LIN {X 0,Y 490.023,Z 695.478,A -85,B 0,C 180,E1 -6692.2,E2 -6692.2} C_VEL
LIN {X 0,Y 489.637,Z 706.697,A -85,B 0,C 180,E1 -6693.054,E2 -6693.054} C_VEL
LIN {X 0,Y 489.247,Z 716.032,A -85,B 0,C 180,E1 -6693.937,E2 -6693.937} C_VEL
LIN {X 0,Y 488.869,Z 726.03,A -85,B 0,C 180,E1 -6695.103,E2 -6695.103} C_VEL
LIN {X 0,Y 488.534,Z 734.515,A -85,B 0,C 180,E1 -6696.331,E2 -6696.331} C_VEL
LIN {X 0,Y 488.289,Z 741.806,A -85,B 0,C 180,E1 -6697.663,E2 -6697.663} C_VEL
LIN {X 0,Y 488.104,Z 747.453,A -85,B 0,C 180,E1 -6698.966,E2 -6698.966} C_VEL
LIN {X 0,Y 487.973,Z 752.212,A -85,B 0,C 180,E1 -6700.399,E2 -6700.399} C_VEL
LIN {X 0,Y 487.929,Z 754.875,A -85,B 0,C 180,E1 -6701.497,E2 -6701.497} C_VEL
LIN {X 0,Y 487.873,Z 756.978,A -85,B 0,C 180,E1 -6702.72,E2 -6702.72} C_VEL
LIN {X 0,Y 487.815,Z 758.178,A -85,B 0,C 180,E1 -6703.916,E2 -6703.916} C_VEL
LIN {X 0,Y 487.843,Z 758.558,A -85,B 0,C 180,E1 -6705.097,E2 -6705.097} C_VEL
LIN {X 0,Y 487.798,Z 758.129,A -85,B 0,C 180,E1 -6706.246,E2 -6706.246} C_VEL
LIN {X 0,Y 487.859,Z 756.943,A -85,B 0,C 180,E1 -6707.385,E2 -6707.385} C_VEL
LIN {X 0,Y 487.942,Z 753.839,A -85,B 0,C 180,E1 -6709.053,E2 -6709.053} C_VEL
LIN {X 0,Y 488.009,Z 750.6,A -85,B 0,C 180,E1 -6710.221,E2 -6710.221} C_VEL
LIN {X 0,Y 488.153,Z 746.364,A -85,B 0,C 180,E1 -6711.396,E2 -6711.396} C_VEL
LIN {X 0,Y 488.318,Z 739.847,A -85,B 0,C 180,E1 -6712.809,E2 -6712.809} C_VEL
LIN {X 0,Y 488.606,Z 732.16,A -85,B 0,C 180,E1 -6714.116,E2 -6714.116} C_VEL
LIN {X 0,Y 488.927,Z 724.156,A -85,B 0,C 180,E1 -6715.219,E2 -6715.219} C_VEL
LIN {X 0,Y 489.04,Z 721.727,A -85,B 0,C 180,E1 -6715.512,E2 -6715.512} C_VEL
LIN {X 0,Y 488.548,Z 717.585,A -85,B 0,C 180,E1 -6715.998,E2 -6715.998} C_VEL
LIN {X 0,Y 486.035,Z 710.622,A -85,B 0,C 180,E1 -6716.77,E2 -6716.77} C_VEL
LIN {X 0,Y 483.52,Z 703.21,A -85,B 0,C 180,E1 -6717.488,E2 -6717.488} C_VEL
LIN {X 0,Y 483.027,Z 698.288,A -85,B 0,C 180,E1 -6717.882,E2 -6717.882} C_VEL
LIN {X 0,Y 483.462,Z 686.391,A -85,B 0,C 180,E1 -6718.646,E2 -6718.646} C_VEL
LIN {X 0,Y 483.818,Z 674.44,A -85,B 0,C 180,E1 -6719.224,E2 -6719.224} C_VEL
LIN {X 0,Y 483.703,Z 669.212,A -85,B 0,C 180,E1 -6719.433,E2 -6719.433} C_VEL
LIN {X 0,Y 481.382,Z 657.052,A -85,B 0,C 180,E1 -6719.872,E2 -6719.872} C_VEL
LIN {X 0,Y 480.883,Z 654.653,A -85,B 0,C 180,E1 -6719.948,E2 -6719.948} C_VEL
LIN {X 0,Y 480.973,Z 649.74,A -85,B 0,C 180,E1 -6723.065,E2 -6723.065} C_VEL
LIN {X 0,Y 481.009,Z 645.406,A -85,B 0,C 180,E1 -6725.851,E2 -6725.851} C_VEL
LIN {X 0,Y 481.143,Z 641.233,A -85,B 0,C 180,E1 -6728.582,E2 -6728.582} C_VEL
LIN {X 0,Y 481.289,Z 636.602,A -85,B 0,C 180,E1 -6731.652,E2 -6731.652} C_VEL
LIN {X 0,Y 481.411,Z 632.002,A -85,B 0,C 180,E1 -6734.765,E2 -6734.765} C_VEL
LIN {X 0,Y 481.586,Z 627.011,A -85,B 0,C 180,E1 -6738.211,E2 -6738.211} C_VEL
LIN {X 0,Y 481.544,Z 624.616,A -85,B 0,C 180,E1 -6739.913,E2 -6739.913} C_VEL
LIN {X 0,Y 481.85,Z 624.467,A -85,B 0,C 180,E1 -6742.664,E2 -6742.664} C_VEL
LIN {X 0,Y 481.783,Z 624.475,A -85,B 0,C 180,E1 -6744.978,E2 -6744.978} C_VEL
LIN {X 0,Y 481.932,Z 624.454,A -85,B 0,C 180,E1 -6747.492,E2 -6747.492} C_VEL
LIN {X 0,Y 481.91,Z 624.46,A -85,B 0,C 180,E1 -6750.835,E2 -6750.835} C_VEL
LIN {X 0,Y 481.932,Z 624.455,A -85,B 0,C 180,E1 -6752.507,E2 -6752.507} C_VEL
LIN {X 0,Y 481.811,Z 624.469,A -85,B 0,C 180,E1 -6755.86,E2 -6755.86} C_VEL
LIN {X 0,Y 481.708,Z 624.483,A -85,B 0,C 180,E1 -6758.389,E2 -6758.389} C_VEL
LIN {X 0,Y 481.338,Z 624.586,A -85,B 0,C 180,E1 -6761.154,E2 -6761.154} C_VEL
LIN {X 0,Y 481.208,Z 629.999,A -85,B 0,C 180,E1 -6764.375,E2 -6764.375} C_VEL
LIN {X 0,Y 481.122,Z 634.354,A -85,B 0,C 180,E1 -6766.986,E2 -6766.986} C_VEL
LIN {X 0,Y 481.049,Z 638.759,A -85,B 0,C 180,E1 -6769.634,E2 -6769.634} C_VEL
LIN {X 0,Y 480.996,Z 643.209,A -85,B 0,C 180,E1 -6772.327,E2 -6772.327} C_VEL
LIN {X 0,Y 480.957,Z 647.726,A -85,B 0,C 180,E1 -6775.072,E2 -6775.072} C_VEL
LIN {X 0,Y 480.865,Z 652.373,A -85,B 0,C 180,E1 -6777.884,E2 -6777.884} C_VEL
LIN {X 0,Y 480.892,Z 654.41,A -85,B 0,C 180,E1 -6779.133,E2 -6779.133} C_VEL
LIN {X 0,Y 483.713,Z 669.153,A -85,B 0,C 180,E1 -6779.663,E2 -6779.663} C_VEL
LIN {X 0,Y 483.735,Z 677.755,A -85,B 0,C 180,E1 -6780.021,E2 -6780.021} C_VEL
LIN {X 0,Y 483.363,Z 688.737,A -85,B 0,C 180,E1 -6780.589,E2 -6780.589} C_VEL
LIN {X 0,Y 482.887,Z 700.545,A -85,B 0,C 180,E1 -6781.385,E2 -6781.385} C_VEL
LIN {X 0,Y 482.421,Z 711.603,A -85,B 0,C 180,E1 -6782.332,E2 -6782.332} C_VEL
LIN {X 0,Y 481.997,Z 721.578,A -85,B 0,C 180,E1 -6783.396,E2 -6783.396} C_VEL
LIN {X 0,Y 481.589,Z 731.3,A -85,B 0,C 180,E1 -6784.69,E2 -6784.69} C_VEL
LIN {X 0,Y 481.293,Z 738.762,A -85,B 0,C 180,E1 -6785.94,E2 -6785.94} C_VEL
LIN {X 0,Y 481.113,Z 744.188,A -85,B 0,C 180,E1 -6787.054,E2 -6787.054} C_VEL
LIN {X 0,Y 480.98,Z 749.367,A -85,B 0,C 180,E1 -6788.388,E2 -6788.388} C_VEL
LIN {X 0,Y 480.842,Z 753.003,A -85,B 0,C 180,E1 -6789.598,E2 -6789.598} C_VEL
LIN {X 0,Y 480.715,Z 756.291,A -85,B 0,C 180,E1 -6791.139,E2 -6791.139} C_VEL
LIN {X 0,Y 480.714,Z 757.779,A -85,B 0,C 180,E1 -6792.261,E2 -6792.261} C_VEL
LIN {X 0,Y 480.698,Z 758.562,A -85,B 0,C 180,E1 -6793.405,E2 -6793.405} C_VEL
LIN {X 0,Y 480.749,Z 758.608,A -85,B 0,C 180,E1 -6794.563,E2 -6794.563} C_VEL
LIN {X 0,Y 480.737,Z 757.873,A -85,B 0,C 180,E1 -6795.752,E2 -6795.752} C_VEL
LIN {X 0,Y 480.748,Z 756.287,A -85,B 0,C 180,E1 -6796.965,E2 -6796.965} C_VEL
LIN {X 0,Y 480.85,Z 753.79,A -85,B 0,C 180,E1 -6798.193,E2 -6798.193} C_VEL
LIN {X 0,Y 480.972,Z 750.253,A -85,B 0,C 180,E1 -6799.448,E2 -6799.448} C_VEL
LIN {X 0,Y 481.131,Z 745.519,A -85,B 0,C 180,E1 -6800.73,E2 -6800.73} C_VEL
LIN {X 0,Y 481.281,Z 739.339,A -85,B 0,C 180,E1 -6802.049,E2 -6802.049} C_VEL
LIN {X 0,Y 481.631,Z 731.527,A -85,B 0,C 180,E1 -6803.375,E2 -6803.375} C_VEL
LIN {X 0,Y 481.975,Z 722.802,A -85,B 0,C 180,E1 -6804.555,E2 -6804.555} C_VEL
LIN {X 0,Y 482.375,Z 713.597,A -85,B 0,C 180,E1 -6805.571,E2 -6805.571} C_VEL
LIN {X 0,Y 482.775,Z 704.293,A -85,B 0,C 180,E1 -6806.414,E2 -6806.414} C_VEL
LIN {X 0,Y 483.225,Z 692.734,A -85,B 0,C 180,E1 -6807.258,E2 -6807.258} C_VEL
LIN {X 0,Y 483.693,Z 679.943,A -85,B 0,C 180,E1 -6807.971,E2 -6807.971} C_VEL
LIN {X 0,Y 483.839,Z 670.339,A -85,B 0,C 180,E1 -6808.38,E2 -6808.38} C_VEL
LIN {X 0,Y 481.643,Z 658.099,A -85,B 0,C 180,E1 -6808.832,E2 -6808.832} C_VEL
LIN {X 0,Y 480.9,Z 654.64,A -85,B 0,C 180,E1 -6808.931,E2 -6808.931} C_VEL
LIN {X 0,Y 480.927,Z 649.312,A -85,B 0,C 180,E1 -6812.119,E2 -6812.119} C_VEL
LIN {X 0,Y 480.987,Z 644.59,A -85,B 0,C 180,E1 -6814.946,E2 -6814.946} C_VEL
LIN {X 0,Y 481.024,Z 639.996,A -85,B 0,C 180,E1 -6817.674,E2 -6817.674} C_VEL
LIN {X 0,Y 481.088,Z 635.435,A -85,B 0,C 180,E1 -6820.367,E2 -6820.367} C_VEL
LIN {X 0,Y 481.139,Z 630.754,A -85,B 0,C 180,E1 -6823.014,E2 -6823.014} C_VEL
LIN {X 0,Y 481.185,Z 626.098,A -85,B 0,C 180,E1 -6825.623,E2 -6825.623} C_VEL
LIN {X 0,Y 481.186,Z 624.552,A -85,B 0,C 180,E1 -6826.486,E2 -6826.486} C_VEL
LIN {X 0,Y 481.553,Z 624.504,A -85,B 0,C 180,E1 -6828.21,E2 -6828.21} C_VEL
LIN {X 0,Y 481.729,Z 624.482,A -85,B 0,C 180,E1 -6830.765,E2 -6830.765} C_VEL
LIN {X 0,Y 481.786,Z 624.476,A -85,B 0,C 180,E1 -6833.298,E2 -6833.298} C_VEL
LIN {X 0,Y 481.661,Z 624.49,A -85,B 0,C 180,E1 -6835.816,E2 -6835.816} C_VEL
LIN {X 0,Y 481.926,Z 624.456,A -85,B 0,C 180,E1 -6837.492,E2 -6837.492} C_VEL
LIN {X 0,Y 481.937,Z 624.455,A -85,B 0,C 180,E1 -6840,E2 -6840} C_VEL
LIN {X 0,Y 481.925,Z 624.458,A -85,B 0,C 180,E1 -6842.507,E2 -6842.507} C_VEL
LIN {X 0,Y 481.814,Z 624.47,A -85,B 0,C 180,E1 -6845.86,E2 -6845.86} C_VEL
LIN {X 0,Y 481.761,Z 624.477,A -85,B 0,C 180,E1 -6848.388,E2 -6848.388} C_VEL
LIN {X 0,Y 481.749,Z 624.478,A -85,B 0,C 180,E1 -6851.785,E2 -6851.785} C_VEL
LIN {X 0,Y 481.739,Z 624.479,A -85,B 0,C 180,E1 -6855.224,E2 -6855.224} C_VEL
LIN {X 0,Y 481.709,Z 624.484,A -85,B 0,C 180,E1 -6858.722,E2 -6858.722} C_VEL
LIN {X 0,Y 481.644,Z 624.49,A -85,B 0,C 180,E1 -6861.395,E2 -6861.395} C_VEL
LIN {X 0,Y 481.674,Z 624.488,A -85,B 0,C 180,E1 -6864.113,E2 -6864.113} C_VEL
LIN {X 0,Y 481.749,Z 624.48,A -85,B 0,C 180,E1 -6867.141,E2 -6867.141} C_VEL
LIN {X 0,Y 481.685,Z 624.486,A -85,B 0,C 180,E1 -6869.741,E2 -6869.741} C_VEL
LIN {X 0,Y 481.67,Z 624.487,A -85,B 0,C 180,E1 -6872.674,E2 -6872.674} C_VEL
LIN {X 0,Y 481.639,Z 624.491,A -85,B 0,C 180,E1 -6875.71,E2 -6875.71} C_VEL
LIN {X 0,Y 481.669,Z 624.488,A -85,B 0,C 180,E1 -6878.859,E2 -6878.859} C_VEL
LIN {X 0,Y 481.65,Z 624.489,A -85,B 0,C 180,E1 -6881.913,E2 -6881.913} C_VEL
LIN {X 0,Y 481.657,Z 624.491,A -85,B 0,C 180,E1 -6884.458,E2 -6884.458} C_VEL
LIN {X 0,Y 481.646,Z 624.492,A -85,B 0,C 180,E1 -6887.84,E2 -6887.84} C_VEL
LIN {X 0,Y 481.69,Z 624.487,A -85,B 0,C 180,E1 -6891.198,E2 -6891.198} C_VEL
LIN {X 0,Y 482.525,Z 629.808,A -85,B 0,C 180,E1 -6893.852,E2 -6893.852} C_VEL
LIN {X 0,Y 482.49,Z 634.708,A -85,B 0,C 180,E1 -6896.127,E2 -6896.127} C_VEL
LIN {X 0,Y 482.181,Z 641.908,A -85,B 0,C 180,E1 -6899.327,E2 -6899.327} C_VEL
LIN {X 0,Y 481.924,Z 648.538,A -85,B 0,C 180,E1 -6902.183,E2 -6902.183} C_VEL
LIN {X 0,Y 481.664,Z 656.3,A -85,B 0,C 180,E1 -6905.428,E2 -6905.428} C_VEL
LIN {X 0,Y 481.461,Z 664.091,A -85,B 0,C 180,E1 -6908.597,E2 -6908.597} C_VEL
LIN {X 0,Y 481.272,Z 671.804,A -85,B 0,C 180,E1 -6911.658,E2 -6911.658} C_VEL
LIN {X 0,Y 481.166,Z 680.269,A -85,B 0,C 180,E1 -6914.974,E2 -6914.974} C_VEL
LIN {X 0,Y 481.134,Z 680.479,A -85,B 0,C 180,E1 -6915.055,E2 -6915.055} C_VEL
LIN {X 0,Y 483.566,Z 695.571,A -85,B 0,C 180,E1 -6915.548,E2 -6915.548} C_VEL
LIN {X 0,Y 483.818,Z 699.636,A -85,B 0,C 180,E1 -6915.704,E2 -6915.704} C_VEL
LIN {X 0,Y 483.466,Z 711.311,A -85,B 0,C 180,E1 -6916.23,E2 -6916.23} C_VEL
LIN {X 0,Y 483.038,Z 722.534,A -85,B 0,C 180,E1 -6916.892,E2 -6916.892} C_VEL
LIN {X 0,Y 482.657,Z 733.399,A -85,B 0,C 180,E1 -6917.705,E2 -6917.705} C_VEL
LIN {X 0,Y 482.232,Z 743.634,A -85,B 0,C 180,E1 -6918.654,E2 -6918.654} C_VEL
LIN {X 0,Y 481.818,Z 752.836,A -85,B 0,C 180,E1 -6919.707,E2 -6919.707} C_VEL
LIN {X 0,Y 481.458,Z 761.8,A -85,B 0,C 180,E1 -6920.972,E2 -6920.972} C_VEL
LIN {X 0,Y 481.194,Z 769.017,A -85,B 0,C 180,E1 -6922.236,E2 -6922.236} C_VEL
LIN {X 0,Y 480.982,Z 774.847,A -85,B 0,C 180,E1 -6923.517,E2 -6923.517} C_VEL
LIN {X 0,Y 480.904,Z 779.936,A -85,B 0,C 180,E1 -6924.97,E2 -6924.97} C_VEL
LIN {X 0,Y 480.842,Z 782.235,A -85,B 0,C 180,E1 -6925.809,E2 -6925.809} C_VEL
LIN {X 0,Y 480.891,Z 784.102,A -85,B 0,C 180,E1 -6926.649,E2 -6926.649} C_VEL
LIN {X 0,Y 480.789,Z 786.495,A -85,B 0,C 180,E1 -6928.325,E2 -6928.325} C_VEL
LIN {X 0,Y 480.76,Z 787.101,A -85,B 0,C 180,E1 -6929.163,E2 -6929.163} C_VEL
LIN {X 0,Y 480.743,Z 787.314,A -85,B 0,C 180,E1 -6930,E2 -6930} C_VEL
LIN {X 0,Y 480.76,Z 787.096,A -85,B 0,C 180,E1 -6930.838,E2 -6930.838} C_VEL
LIN {X 0,Y 480.79,Z 786.486,A -85,B 0,C 180,E1 -6931.676,E2 -6931.676} C_VEL
LIN {X 0,Y 480.891,Z 784.082,A -85,B 0,C 180,E1 -6933.352,E2 -6933.352} C_VEL
LIN {X 0,Y 480.853,Z 781.13,A -85,B 0,C 180,E1 -6934.611,E2 -6934.611} C_VEL
LIN {X 0,Y 480.987,Z 777.14,A -85,B 0,C 180,E1 -6935.871,E2 -6935.871} C_VEL
LIN {X 0,Y 481.113,Z 770.999,A -85,B 0,C 180,E1 -6937.344,E2 -6937.344} C_VEL
LIN {X 0,Y 481.362,Z 764.292,A -85,B 0,C 180,E1 -6938.607,E2 -6938.607} C_VEL
LIN {X 0,Y 481.667,Z 755.968,A -85,B 0,C 180,E1 -6939.872,E2 -6939.872} C_VEL
LIN {X 0,Y 482.04,Z 747.432,A -85,B 0,C 180,E1 -6940.926,E2 -6940.926} C_VEL
LIN {X 0,Y 482.547,Z 736.893,A -85,B 0,C 180,E1 -6941.979,E2 -6941.979} C_VEL
LIN {X 0,Y 482.877,Z 725.625,A -85,B 0,C 180,E1 -6942.887,E2 -6942.887} C_VEL
LIN {X 0,Y 483.273,Z 715.042,A -85,B 0,C 180,E1 -6943.562,E2 -6943.562} C_VEL
LIN {X 0,Y 483.716,Z 703.29,A -85,B 0,C 180,E1 -6944.139,E2 -6944.139} C_VEL
LIN {X 0,Y 483.703,Z 696.454,A -85,B 0,C 180,E1 -6944.408,E2 -6944.408} C_VEL
LIN {X 0,Y 481.537,Z 683.152,A -85,B 0,C 180,E1 -6944.859,E2 -6944.859} C_VEL
LIN {X 0,Y 481.122,Z 680.302,A -85,B 0,C 180,E1 -6944.947,E2 -6944.947} C_VEL
LIN {X 0,Y 481.225,Z 672.754,A -85,B 0,C 180,E1 -6947.86,E2 -6947.86} C_VEL
LIN {X 0,Y 481.462,Z 665.027,A -85,B 0,C 180,E1 -6950.897,E2 -6950.897} C_VEL
LIN {X 0,Y 481.642,Z 655.92,A -85,B 0,C 180,E1 -6954.574,E2 -6954.574} C_VEL
LIN {X 0,Y 481.899,Z 648.163,A -85,B 0,C 180,E1 -6957.82,E2 -6957.82} C_VEL
LIN {X 0,Y 482.125,Z 641.589,A -85,B 0,C 180,E1 -6960.677,E2 -6960.677} C_VEL
LIN {X 0,Y 482.421,Z 635.103,A -85,B 0,C 180,E1 -6963.614,E2 -6963.614} C_VEL
LIN {X 0,Y 482.586,Z 630.852,A -85,B 0,C 180,E1 -6965.629,E2 -6965.629} C_VEL
LIN {X 0,Y 481.974,Z 626.099,A -85,B 0,C 180,E1 -6968.056,E2 -6968.056} C_VEL
LIN {X 0,Y 481.678,Z 624.488,A -85,B 0,C 180,E1 -6968.981,E2 -6968.981} C_VEL
LIN {X 0,Y 481.656,Z 624.493,A -85,B 0,C 180,E1 -6972.16,E2 -6972.16} C_VEL
LIN {X 0,Y 481.662,Z 624.49,A -85,B 0,C 180,E1 -6975.543,E2 -6975.543} C_VEL
LIN {X 0,Y 481.658,Z 624.491,A -85,B 0,C 180,E1 -6978.958,E2 -6978.958} C_VEL
LIN {X 0,Y 481.657,Z 624.49,A -85,B 0,C 180,E1 -6981.993,E2 -6981.993} C_VEL
LIN {X 0,Y 481.693,Z 624.487,A -85,B 0,C 180,E1 -6985.318,E2 -6985.318} C_VEL
LIN {X 0,Y 481.647,Z 624.491,A -85,B 0,C 180,E1 -6988.312,E2 -6988.312} C_VEL
LIN {X 0,Y 481.702,Z 624.485,A -85,B 0,C 180,E1 -6991.219,E2 -6991.219} C_VEL
LIN {X 0,Y 481.703,Z 624.483,A -85,B 0,C 180,E1 -6994.043,E2 -6994.043} C_VEL
LIN {X 0,Y 481.676,Z 624.488,A -85,B 0,C 180,E1 -6996.812,E2 -6996.812} C_VEL
LIN {X 0,Y 481.699,Z 624.486,A -85,B 0,C 180,E1 -6999.503,E2 -6999.503} C_VEL
LIN {X 0,Y 481.709,Z 624.483,A -85,B 0,C 180,E1 -7002.159,E2 -7002.159} C_VEL
LIN {X 0,Y 481.744,Z 624.479,A -85,B 0,C 180,E1 -7004.776,E2 -7004.776} C_VEL
LIN {X 0,Y 481.752,Z 624.478,A -85,B 0,C 180,E1 -7008.215,E2 -7008.215} C_VEL
LIN {X 0,Y 481.765,Z 624.478,A -85,B 0,C 180,E1 -7011.612,E2 -7011.612} C_VEL
LIN {X 0,Y 481.818,Z 624.469,A -85,B 0,C 180,E1 -7014.14,E2 -7014.14} C_VEL
LIN {X 0,Y 481.929,Z 624.456,A -85,B 0,C 180,E1 -7017.493,E2 -7017.493} C_VEL
LIN {X 0,Y 481.908,Z 624.461,A -85,B 0,C 180,E1 -7020.836,E2 -7020.836} C_VEL
LIN {X 0,Y 481.93,Z 624.457,A -85,B 0,C 180,E1 -7022.507,E2 -7022.507} C_VEL
LIN {X 0,Y 481.819,Z 624.471,A -85,B 0,C 180,E1 -7025.86,E2 -7025.86} C_VEL
LIN {X 0,Y 481.749,Z 624.48,A -85,B 0,C 180,E1 -7028.389,E2 -7028.389} C_VEL
LIN {X 0,Y 481.696,Z 624.487,A -85,B 0,C 180,E1 -7029.235,E2 -7029.235} C_VEL
LIN {X 0,Y 481.635,Z 626.43,A -85,B 0,C 180,E1 -7030.935,E2 -7030.935} C_VEL
LIN {X 0,Y 481.49,Z 630.017,A -85,B 0,C 180,E1 -7033.506,E2 -7033.506} C_VEL
LIN {X 0,Y 481.397,Z 633.712,A -85,B 0,C 180,E1 -7036.104,E2 -7036.104} C_VEL
LIN {X 0,Y 481.29,Z 637.531,A -85,B 0,C 180,E1 -7038.739,E2 -7038.739} C_VEL
LIN {X 0,Y 481.181,Z 641.484,A -85,B 0,C 180,E1 -7041.417,E2 -7041.417} C_VEL
LIN {X 0,Y 481.073,Z 645.608,A -85,B 0,C 180,E1 -7044.145,E2 -7044.145} C_VEL
LIN {X 0,Y 481.013,Z 649.913,A -85,B 0,C 180,E1 -7046.968,E2 -7046.968} C_VEL
LIN {X 0,Y 480.901,Z 654.887,A -85,B 0,C 180,E1 -7050.147,E2 -7050.147} C_VEL
LIN {X 0,Y 483.356,Z 666.994,A -85,B 0,C 180,E1 -7050.562,E2 -7050.562} C_VEL
LIN {X 0,Y 483.926,Z 670.742,A -85,B 0,C 180,E1 -7050.714,E2 -7050.714} C_VEL
LIN {X 0,Y 483.599,Z 683.35,A -85,B 0,C 180,E1 -7051.278,E2 -7051.278} C_VEL
LIN {X 0,Y 483.139,Z 694.659,A -85,B 0,C 180,E1 -7051.947,E2 -7051.947} C_VEL
LIN {X 0,Y 482.701,Z 706.476,A -85,B 0,C 180,E1 -7052.844,E2 -7052.844} C_VEL
LIN {X 0,Y 482.255,Z 716.754,A -85,B 0,C 180,E1 -7053.832,E2 -7053.832} C_VEL
LIN {X 0,Y 481.894,Z 726.063,A -85,B 0,C 180,E1 -7054.936,E2 -7054.936} C_VEL
LIN {X 0,Y 481.522,Z 734.363,A -85,B 0,C 180,E1 -7056.145,E2 -7056.145} C_VEL
LIN {X 0,Y 481.251,Z 740.817,A -85,B 0,C 180,E1 -7057.305,E2 -7057.305} C_VEL
LIN {X 0,Y 481.063,Z 746.823,A -85,B 0,C 180,E1 -7058.656,E2 -7058.656} C_VEL
LIN {X 0,Y 480.922,Z 751.496,A -85,B 0,C 180,E1 -7060.016,E2 -7060.016} C_VEL
LIN {X 0,Y 480.87,Z 754.408,A -85,B 0,C 180,E1 -7061.124,E2 -7061.124} C_VEL
LIN {X 0,Y 480.777,Z 756.578,A -85,B 0,C 180,E1 -7062.255,E2 -7062.255} C_VEL
LIN {X 0,Y 480.712,Z 758,A -85,B 0,C 180,E1 -7063.404,E2 -7063.404} C_VEL
LIN {X 0,Y 480.75,Z 758.69,A -85,B 0,C 180,E1 -7064.564,E2 -7064.564} C_VEL
LIN {X 0,Y 480.741,Z 758.628,A -85,B 0,C 180,E1 -7065.753,E2 -7065.753} C_VEL
LIN {X 0,Y 480.735,Z 757.715,A -85,B 0,C 180,E1 -7066.968,E2 -7066.968} C_VEL
LIN {X 0,Y 480.807,Z 755.924,A -85,B 0,C 180,E1 -7068.2,E2 -7068.2} C_VEL
LIN {X 0,Y 480.895,Z 753.164,A -85,B 0,C 180,E1 -7069.46,E2 -7069.46} C_VEL
LIN {X 0,Y 480.999,Z 749.288,A -85,B 0,C 180,E1 -7070.751,E2 -7070.751} C_VEL
LIN {X 0,Y 481.17,Z 743.729,A -85,B 0,C 180,E1 -7072.16,E2 -7072.16} C_VEL
LIN {X 0,Y 481.369,Z 737.385,A -85,B 0,C 180,E1 -7073.418,E2 -7073.418} C_VEL
LIN {X 0,Y 481.656,Z 730.209,A -85,B 0,C 180,E1 -7074.571,E2 -7074.571} C_VEL
LIN {X 0,Y 482.086,Z 720.825,A -85,B 0,C 180,E1 -7075.793,E2 -7075.793} C_VEL
LIN {X 0,Y 482.47,Z 711.662,A -85,B 0,C 180,E1 -7076.765,E2 -7076.765} C_VEL
LIN {X 0,Y 482.919,Z 701.18,A -85,B 0,C 180,E1 -7077.668,E2 -7077.668} C_VEL
LIN {X 0,Y 483.027,Z 698.288,A -85,B 0,C 180,E1 -7077.882,E2 -7077.882} C_VEL
LIN {X 0,Y 482.387,Z 691.624,A -85,B 0,C 180,E1 -7078.37,E2 -7078.37} C_VEL
LIN {X 0,Y 480.649,Z 684.948,A -85,B 0,C 180,E1 -7078.826,E2 -7078.826} C_VEL
LIN {X 0,Y 477.659,Z 674.561,A -85,B 0,C 180,E1 -7079.42,E2 -7079.42} C_VEL
LIN {X 0,Y 476.946,Z 670.914,A -85,B 0,C 180,E1 -7079.584,E2 -7079.584} C_VEL
LIN {X 0,Y 474.785,Z 659.451,A -85,B 0,C 180,E1 -7080.027,E2 -7080.027} C_VEL
LIN {X 0,Y 473.821,Z 654.8,A -85,B 0,C 180,E1 -7080.19,E2 -7080.19} C_VEL
LIN {X 0,Y 473.894,Z 649.522,A -85,B 0,C 180,E1 -7083.582,E2 -7083.582} C_VEL
LIN {X 0,Y 474.02,Z 644.577,A -85,B 0,C 180,E1 -7086.815,E2 -7086.815} C_VEL
LIN {X 0,Y 474.134,Z 639.695,A -85,B 0,C 180,E1 -7090.067,E2 -7090.067} C_VEL
LIN {X 0,Y 474.238,Z 635.713,A -85,B 0,C 180,E1 -7092.759,E2 -7092.759} C_VEL
LIN {X 0,Y 474.344,Z 631.858,A -85,B 0,C 180,E1 -7095.411,E2 -7095.411} C_VEL
LIN {X 0,Y 474.533,Z 628.115,A -85,B 0,C 180,E1 -7098.033,E2 -7098.033} C_VEL
LIN {X 0,Y 474.496,Z 625.698,A -85,B 0,C 180,E1 -7099.762,E2 -7099.762} C_VEL
LIN {X 0,Y 474.696,Z 625.355,A -85,B 0,C 180,E1 -7101.486,E2 -7101.486} C_VEL
LIN {X 0,Y 474.781,Z 625.345,A -85,B 0,C 180,E1 -7104.052,E2 -7104.052} C_VEL
LIN {X 0,Y 474.898,Z 625.33,A -85,B 0,C 180,E1 -7107.455,E2 -7107.455} C_VEL
LIN {X 0,Y 474.916,Z 625.328,A -85,B 0,C 180,E1 -7110,E2 -7110} C_VEL
LIN {X 0,Y 474.898,Z 625.331,A -85,B 0,C 180,E1 -7112.544,E2 -7112.544} C_VEL
LIN {X 0,Y 474.773,Z 625.345,A -85,B 0,C 180,E1 -7115.947,E2 -7115.947} C_VEL
LIN {X 0,Y 474.649,Z 625.362,A -85,B 0,C 180,E1 -7118.515,E2 -7118.515} C_VEL
LIN {X 0,Y 474.298,Z 625.578,A -85,B 0,C 180,E1 -7121.321,E2 -7121.321} C_VEL
LIN {X 0,Y 474.144,Z 631.031,A -85,B 0,C 180,E1 -7124.594,E2 -7124.594} C_VEL
LIN {X 0,Y 474.04,Z 635.44,A -85,B 0,C 180,E1 -7127.248,E2 -7127.248} C_VEL
LIN {X 0,Y 473.958,Z 639.867,A -85,B 0,C 180,E1 -7129.94,E2 -7129.94} C_VEL
LIN {X 0,Y 473.907,Z 645.152,A -85,B 0,C 180,E1 -7133.153,E2 -7133.153} C_VEL
LIN {X 0,Y 473.866,Z 648.952,A -85,B 0,C 180,E1 -7135.474,E2 -7135.474} C_VEL
LIN {X 0,Y 473.803,Z 654.587,A -85,B 0,C 180,E1 -7138.921,E2 -7138.921} C_VEL
LIN {X 0,Y 476.566,Z 668.419,A -85,B 0,C 180,E1 -7139.412,E2 -7139.412} C_VEL
LIN {X 0,Y 476.994,Z 673.44,A -85,B 0,C 180,E1 -7139.622,E2 -7139.622} C_VEL
LIN {X 0,Y 476.52,Z 685.823,A -85,B 0,C 180,E1 -7140.218,E2 -7140.218} C_VEL
LIN {X 0,Y 476.071,Z 698.305,A -85,B 0,C 180,E1 -7141.018,E2 -7141.018} C_VEL
LIN {X 0,Y 475.63,Z 708.873,A -85,B 0,C 180,E1 -7141.887,E2 -7141.887} C_VEL
LIN {X 0,Y 475.205,Z 718.224,A -85,B 0,C 180,E1 -7142.833,E2 -7142.833} C_VEL
LIN {X 0,Y 474.723,Z 727.63,A -85,B 0,C 180,E1 -7143.999,E2 -7143.999} C_VEL
LIN {X 0,Y 474.372,Z 736.052,A -85,B 0,C 180,E1 -7145.295,E2 -7145.295} C_VEL
LIN {X 0,Y 474.084,Z 743.825,A -85,B 0,C 180,E1 -7146.82,E2 -7146.82} C_VEL
LIN {X 0,Y 473.932,Z 749.19,A -85,B 0,C 180,E1 -7148.192,E2 -7148.192} C_VEL
LIN {X 0,Y 473.765,Z 753.457,A -85,B 0,C 180,E1 -7149.633,E2 -7149.633} C_VEL
LIN {X 0,Y 473.656,Z 756.016,A -85,B 0,C 180,E1 -7150.823,E2 -7150.823} C_VEL
LIN {X 0,Y 473.618,Z 757.846,A -85,B 0,C 180,E1 -7152.102,E2 -7152.102} C_VEL
LIN {X 0,Y 473.602,Z 758.756,A -85,B 0,C 180,E1 -7153.353,E2 -7153.353} C_VEL
LIN {X 0,Y 473.652,Z 758.813,A -85,B 0,C 180,E1 -7154.584,E2 -7154.584} C_VEL
LIN {X 0,Y 473.64,Z 758.073,A -85,B 0,C 180,E1 -7155.781,E2 -7155.781} C_VEL
LIN {X 0,Y 473.652,Z 756.572,A -85,B 0,C 180,E1 -7156.957,E2 -7156.957} C_VEL
LIN {X 0,Y 473.764,Z 754.315,A -85,B 0,C 180,E1 -7158.122,E2 -7158.122} C_VEL
LIN {X 0,Y 473.877,Z 751.306,A -85,B 0,C 180,E1 -7159.265,E2 -7159.265} C_VEL
LIN {X 0,Y 474.039,Z 746.204,A -85,B 0,C 180,E1 -7160.713,E2 -7160.713} C_VEL
LIN {X 0,Y 474.218,Z 740.52,A -85,B 0,C 180,E1 -7161.974,E2 -7161.974} C_VEL
LIN {X 0,Y 474.468,Z 734.184,A -85,B 0,C 180,E1 -7163.116,E2 -7163.116} C_VEL
LIN {X 0,Y 474.821,Z 725.924,A -85,B 0,C 180,E1 -7164.334,E2 -7164.334} C_VEL
LIN {X 0,Y 475.314,Z 716.771,A -85,B 0,C 180,E1 -7165.43,E2 -7165.43} C_VEL
LIN {X 0,Y 475.701,Z 707.268,A -85,B 0,C 180,E1 -7166.356,E2 -7166.356} C_VEL
LIN {X 0,Y 476.202,Z 695.6,A -85,B 0,C 180,E1 -7167.269,E2 -7167.269} C_VEL
LIN {X 0,Y 476.693,Z 683.456,A -85,B 0,C 180,E1 -7168.005,E2 -7168.005} C_VEL
LIN {X 0,Y 476.882,Z 670.827,A -85,B 0,C 180,E1 -7168.578,E2 -7168.578} C_VEL
LIN {X 0,Y 474.719,Z 658.959,A -85,B 0,C 180,E1 -7169.031,E2 -7169.031} C_VEL
LIN {X 0,Y 473.817,Z 654.766,A -85,B 0,C 180,E1 -7169.164,E2 -7169.164} C_VEL
LIN {X 0,Y 473.834,Z 650.63,A -85,B 0,C 180,E1 -7171.665,E2 -7171.665} C_VEL
LIN {X 0,Y 473.911,Z 645.481,A -85,B 0,C 180,E1 -7174.77,E2 -7174.77} C_VEL
LIN {X 0,Y 473.946,Z 641.256,A -85,B 0,C 180,E1 -7177.322,E2 -7177.322} C_VEL
LIN {X 0,Y 474.004,Z 636.587,A -85,B 0,C 180,E1 -7180.061,E2 -7180.061} C_VEL
LIN {X 0,Y 474.058,Z 631.898,A -85,B 0,C 180,E1 -7182.752,E2 -7182.752} C_VEL
LIN {X 0,Y 474.147,Z 627.201,A -85,B 0,C 180,E1 -7185.405,E2 -7185.405} C_VEL
LIN {X 0,Y 474.142,Z 625.429,A -85,B 0,C 180,E1 -7186.499,E2 -7186.499} C_VEL
LIN {X 0,Y 474.569,Z 625.375,A -85,B 0,C 180,E1 -7188.9,E2 -7188.9} C_VEL
LIN {X 0,Y 474.723,Z 625.354,A -85,B 0,C 180,E1 -7191.486,E2 -7191.486} C_VEL
LIN {X 0,Y 474.776,Z 625.349,A -85,B 0,C 180,E1 -7194.052,E2 -7194.052} C_VEL
LIN {X 0,Y 474.892,Z 625.333,A -85,B 0,C 180,E1 -7197.455,E2 -7197.455} C_VEL
LIN {X 0,Y 474.874,Z 625.335,A -85,B 0,C 180,E1 -7200.848,E2 -7200.848} C_VEL
LIN {X 0,Y 474.891,Z 625.334,A -85,B 0,C 180,E1 -7202.545,E2 -7202.545} C_VEL
LIN {X 0,Y 474.776,Z 625.346,A -85,B 0,C 180,E1 -7205.948,E2 -7205.948} C_VEL
LIN {X 0,Y 474.726,Z 625.355,A -85,B 0,C 180,E1 -7208.514,E2 -7208.514} C_VEL
LIN {X 0,Y 474.702,Z 625.355,A -85,B 0,C 180,E1 -7211.962,E2 -7211.962} C_VEL
LIN {X 0,Y 474.696,Z 625.357,A -85,B 0,C 180,E1 -7215.456,E2 -7215.456} C_VEL
LIN {X 0,Y 474.662,Z 625.361,A -85,B 0,C 180,E1 -7219.01,E2 -7219.01} C_VEL
LIN {X 0,Y 474.586,Z 625.369,A -85,B 0,C 180,E1 -7221.729,E2 -7221.729} C_VEL
LIN {X 0,Y 474.656,Z 625.361,A -85,B 0,C 180,E1 -7224.493,E2 -7224.493} C_VEL
LIN {X 0,Y 474.696,Z 625.357,A -85,B 0,C 180,E1 -7227.339,E2 -7227.339} C_VEL
LIN {X 0,Y 474.607,Z 625.367,A -85,B 0,C 180,E1 -7230.812,E2 -7230.812} C_VEL
LIN {X 0,Y 474.635,Z 625.364,A -85,B 0,C 180,E1 -7233.984,E2 -7233.984} C_VEL
LIN {X 0,Y 474.571,Z 625.372,A -85,B 0,C 180,E1 -7236.9,E2 -7236.9} C_VEL
LIN {X 0,Y 474.625,Z 625.365,A -85,B 0,C 180,E1 -7239.648,E2 -7239.648} C_VEL
LIN {X 0,Y 474.612,Z 625.367,A -85,B 0,C 180,E1 -7242.935,E2 -7242.935} C_VEL
LIN {X 0,Y 474.608,Z 625.368,A -85,B 0,C 180,E1 -7245.896,E2 -7245.896} C_VEL
LIN {X 0,Y 474.626,Z 625.366,A -85,B 0,C 180,E1 -7249.041,E2 -7249.041} C_VEL
LIN {X 0,Y 474.676,Z 625.46,A -85,B 0,C 180,E1 -7251.074,E2 -7251.074} C_VEL
LIN {X 0,Y 475.51,Z 630.814,A -85,B 0,C 180,E1 -7253.759,E2 -7253.759} C_VEL
LIN {X 0,Y 475.511,Z 635.255,A -85,B 0,C 180,E1 -7255.861,E2 -7255.861} C_VEL
LIN {X 0,Y 475.171,Z 642.353,A -85,B 0,C 180,E1 -7259.076,E2 -7259.076} C_VEL
LIN {X 0,Y 474.884,Z 649.525,A -85,B 0,C 180,E1 -7262.214,E2 -7262.214} C_VEL
LIN {X 0,Y 474.614,Z 657.291,A -85,B 0,C 180,E1 -7265.505,E2 -7265.505} C_VEL
LIN {X 0,Y 474.391,Z 665.65,A -85,B 0,C 180,E1 -7268.961,E2 -7268.961} C_VEL
LIN {X 0,Y 474.159,Z 673.971,A -85,B 0,C 180,E1 -7272.311,E2 -7272.311} C_VEL
LIN {X 0,Y 474.074,Z 680.332,A -85,B 0,C 180,E1 -7274.84,E2 -7274.84} C_VEL
LIN {X 0,Y 476.305,Z 694.158,A -85,B 0,C 180,E1 -7275.282,E2 -7275.282} C_VEL
LIN {X 0,Y 476.924,Z 699.384,A -85,B 0,C 180,E1 -7275.493,E2 -7275.493} C_VEL
LIN {X 0,Y 476.561,Z 711.063,A -85,B 0,C 180,E1 -7276.026,E2 -7276.026} C_VEL
LIN {X 0,Y 476.075,Z 723.401,A -85,B 0,C 180,E1 -7276.773,E2 -7276.773} C_VEL
LIN {X 0,Y 475.651,Z 734.695,A -85,B 0,C 180,E1 -7277.652,E2 -7277.652} C_VEL
LIN {X 0,Y 475.161,Z 745.364,A -85,B 0,C 180,E1 -7278.699,E2 -7278.699} C_VEL
LIN {X 0,Y 474.706,Z 754.242,A -85,B 0,C 180,E1 -7279.767,E2 -7279.767} C_VEL
LIN {X 0,Y 474.362,Z 762.909,A -85,B 0,C 180,E1 -7281.051,E2 -7281.051} C_VEL
LIN {X 0,Y 474.07,Z 769.828,A -85,B 0,C 180,E1 -7282.333,E2 -7282.333} C_VEL
LIN {X 0,Y 473.888,Z 775.087,A -85,B 0,C 180,E1 -7283.539,E2 -7283.539} C_VEL
LIN {X 0,Y 473.838,Z 779.724,A -85,B 0,C 180,E1 -7284.895,E2 -7284.895} C_VEL
LIN {X 0,Y 473.748,Z 782.024,A -85,B 0,C 180,E1 -7285.747,E2 -7285.747} C_VEL
LIN {X 0,Y 473.798,Z 783.892,A -85,B 0,C 180,E1 -7286.599,E2 -7286.599} C_VEL
LIN {X 0,Y 473.695,Z 786.285,A -85,B 0,C 180,E1 -7288.3,E2 -7288.3} C_VEL
LIN {X 0,Y 473.688,Z 786.891,A -85,B 0,C 180,E1 -7289.15,E2 -7289.15} C_VEL
LIN {X 0,Y 473.669,Z 787.104,A -85,B 0,C 180,E1 -7290,E2 -7290} C_VEL
LIN {X 0,Y 473.688,Z 786.885,A -85,B 0,C 180,E1 -7290.85,E2 -7290.85} C_VEL
LIN {X 0,Y 473.724,Z 785.269,A -85,B 0,C 180,E1 -7292.551,E2 -7292.551} C_VEL
LIN {X 0,Y 473.799,Z 783.865,A -85,B 0,C 180,E1 -7293.402,E2 -7293.402} C_VEL
LIN {X 0,Y 473.774,Z 780.909,A -85,B 0,C 180,E1 -7294.68,E2 -7294.68} C_VEL
LIN {X 0,Y 473.876,Z 776.029,A -85,B 0,C 180,E1 -7296.198,E2 -7296.198} C_VEL
LIN {X 0,Y 474.071,Z 769.748,A -85,B 0,C 180,E1 -7297.668,E2 -7297.668} C_VEL
LIN {X 0,Y 474.348,Z 762.807,A -85,B 0,C 180,E1 -7298.95,E2 -7298.95} C_VEL
LIN {X 0,Y 474.693,Z 754.118,A -85,B 0,C 180,E1 -7300.234,E2 -7300.234} C_VEL
LIN {X 0,Y 475.132,Z 745.215,A -85,B 0,C 180,E1 -7301.303,E2 -7301.303} C_VEL
LIN {X 0,Y 475.626,Z 734.571,A -85,B 0,C 180,E1 -7302.344,E2 -7302.344} C_VEL
LIN {X 0,Y 475.998,Z 723.824,A -85,B 0,C 180,E1 -7303.186,E2 -7303.186} C_VEL
LIN {X 0,Y 476.439,Z 712.802,A -85,B 0,C 180,E1 -7303.869,E2 -7303.869} C_VEL
LIN {X 0,Y 476.898,Z 700.41,A -85,B 0,C 180,E1 -7304.454,E2 -7304.454} C_VEL
LIN {X 0,Y 476.278,Z 694.25,A -85,B 0,C 180,E1 -7304.706,E2 -7304.706} C_VEL
LIN {X 0,Y 474.187,Z 681.259,A -85,B 0,C 180,E1 -7305.129,E2 -7305.129} C_VEL
LIN {X 0,Y 474.082,Z 679.996,A -85,B 0,C 180,E1 -7305.201,E2 -7305.201} C_VEL
LIN {X 0,Y 474.191,Z 671.728,A -85,B 0,C 180,E1 -7308.459,E2 -7308.459} C_VEL
LIN {X 0,Y 474.384,Z 665.303,A -85,B 0,C 180,E1 -7311.037,E2 -7311.037} C_VEL
LIN {X 0,Y 474.566,Z 656.869,A -85,B 0,C 180,E1 -7314.498,E2 -7314.498} C_VEL
LIN {X 0,Y 474.863,Z 649.128,A -85,B 0,C 180,E1 -7317.788,E2 -7317.788} C_VEL
LIN {X 0,Y 475.163,Z 641.508,A -85,B 0,C 180,E1 -7321.177,E2 -7321.177} C_VEL
LIN {X 0,Y 475.48,Z 635.064,A -85,B 0,C 180,E1 -7324.172,E2 -7324.172} C_VEL
LIN {X 0,Y 475.477,Z 630.836,A -85,B 0,C 180,E1 -7326.245,E2 -7326.245} C_VEL
LIN {X 0,Y 474.653,Z 625.364,A -85,B 0,C 180,E1 -7329.202,E2 -7329.202} C_VEL
LIN {X 0,Y 474.633,Z 625.367,A -85,B 0,C 180,E1 -7332.238,E2 -7332.238} C_VEL
LIN {X 0,Y 474.623,Z 625.368,A -85,B 0,C 180,E1 -7335.297,E2 -7335.297} C_VEL
LIN {X 0,Y 474.623,Z 625.368,A -85,B 0,C 180,E1 -7338.215,E2 -7338.215} C_VEL
LIN {X 0,Y 474.646,Z 625.365,A -85,B 0,C 180,E1 -7340.454,E2 -7340.454} C_VEL
LIN {X 0,Y 474.592,Z 625.371,A -85,B 0,C 180,E1 -7343.677,E2 -7343.677} C_VEL
LIN {X 0,Y 474.645,Z 625.363,A -85,B 0,C 180,E1 -7346.78,E2 -7346.78} C_VEL
LIN {X 0,Y 474.607,Z 625.367,A -85,B 0,C 180,E1 -7349.77,E2 -7349.77} C_VEL
LIN {X 0,Y 474.699,Z 625.357,A -85,B 0,C 180,E1 -7352.68,E2 -7352.68} C_VEL
LIN {X 0,Y 474.661,Z 625.361,A -85,B 0,C 180,E1 -7355.507,E2 -7355.507} C_VEL
LIN {X 0,Y 474.672,Z 625.359,A -85,B 0,C 180,E1 -7359.185,E2 -7359.185} C_VEL
LIN {X 0,Y 474.659,Z 625.362,A -85,B 0,C 180,E1 -7361.884,E2 -7361.884} C_VEL
LIN {X 0,Y 474.702,Z 625.358,A -85,B 0,C 180,E1 -7364.544,E2 -7364.544} C_VEL
LIN {X 0,Y 474.706,Z 625.356,A -85,B 0,C 180,E1 -7368.038,E2 -7368.038} C_VEL
LIN {X 0,Y 474.73,Z 625.354,A -85,B 0,C 180,E1 -7371.487,E2 -7371.487} C_VEL
LIN {X 0,Y 474.78,Z 625.345,A -85,B 0,C 180,E1 -7374.052,E2 -7374.052} C_VEL
LIN {X 0,Y 474.895,Z 625.332,A -85,B 0,C 180,E1 -7377.455,E2 -7377.455} C_VEL
LIN {X 0,Y 474.913,Z 625.33,A -85,B 0,C 180,E1 -7380,E2 -7380} C_VEL
LIN {X 0,Y 474.896,Z 625.334,A -85,B 0,C 180,E1 -7382.545,E2 -7382.545} C_VEL
LIN {X 0,Y 474.781,Z 625.348,A -85,B 0,C 180,E1 -7385.948,E2 -7385.948} C_VEL
LIN {X 0,Y 474.713,Z 625.356,A -85,B 0,C 180,E1 -7388.514,E2 -7388.514} C_VEL
LIN {X 0,Y 474.63,Z 625.367,A -85,B 0,C 180,E1 -7389.374,E2 -7389.374} C_VEL
LIN {X 0,Y 474.565,Z 629.107,A -85,B 0,C 180,E1 -7392.2,E2 -7392.2} C_VEL
LIN {X 0,Y 474.394,Z 633.897,A -85,B 0,C 180,E1 -7395.644,E2 -7395.644} C_VEL
LIN {X 0,Y 474.224,Z 638.758,A -85,B 0,C 180,E1 -7399.029,E2 -7399.029} C_VEL
LIN {X 0,Y 474.103,Z 642.735,A -85,B 0,C 180,E1 -7401.752,E2 -7401.752} C_VEL
LIN {X 0,Y 473.998,Z 647.955,A -85,B 0,C 180,E1 -7405.251,E2 -7405.251} C_VEL
LIN {X 0,Y 473.874,Z 652.653,A -85,B 0,C 180,E1 -7408.333,E2 -7408.333} C_VEL
LIN {X 0,Y 473.83,Z 655.093,A -85,B 0,C 180,E1 -7409.917,E2 -7409.917} C_VEL
LIN {X 0,Y 476.552,Z 668.434,A -85,B 0,C 180,E1 -7410.398,E2 -7410.398} C_VEL
LIN {X 0,Y 477.035,Z 672.345,A -85,B 0,C 180,E1 -7410.56,E2 -7410.56} C_VEL
LIN {X 0,Y 476.663,Z 684.604,A -85,B 0,C 180,E1 -7411.133,E2 -7411.133} C_VEL
LIN {X 0,Y 476.169,Z 696.448,A -85,B 0,C 180,E1 -7411.863,E2 -7411.863} C_VEL
LIN {X 0,Y 475.736,Z 707.133,A -85,B 0,C 180,E1 -7412.705,E2 -7412.705} C_VEL
LIN {X 0,Y 475.275,Z 717.057,A -85,B 0,C 180,E1 -7413.678,E2 -7413.678} C_VEL
LIN {X 0,Y 474.868,Z 726.857,A -85,B 0,C 180,E1 -7414.865,E2 -7414.865} C_VEL
LIN {X 0,Y 474.461,Z 735.118,A -85,B 0,C 180,E1 -7416.105,E2 -7416.105} C_VEL
LIN {X 0,Y 474.199,Z 742.111,A -85,B 0,C 180,E1 -7417.42,E2 -7417.42} C_VEL
LIN {X 0,Y 474.003,Z 746.863,A -85,B 0,C 180,E1 -7418.516,E2 -7418.516} C_VEL
LIN {X 0,Y 473.893,Z 750.757,A -85,B 0,C 180,E1 -7419.621,E2 -7419.621} C_VEL
LIN {X 0,Y 473.765,Z 755.17,A -85,B 0,C 180,E1 -7421.33,E2 -7421.33} C_VEL
LIN {X 0,Y 473.689,Z 756.618,A -85,B 0,C 180,E1 -7422.112,E2 -7422.112} C_VEL
LIN {X 0,Y 473.619,Z 758.189,A -85,B 0,C 180,E1 -7423.355,E2 -7423.355} C_VEL
LIN {X 0,Y 473.652,Z 758.907,A -85,B 0,C 180,E1 -7424.584,E2 -7424.584} C_VEL
LIN {X 0,Y 473.642,Z 758.83,A -85,B 0,C 180,E1 -7425.781,E2 -7425.781} C_VEL
LIN {X 0,Y 473.638,Z 757.962,A -85,B 0,C 180,E1 -7426.956,E2 -7426.956} C_VEL
LIN {X 0,Y 473.724,Z 756.35,A -85,B 0,C 180,E1 -7428.117,E2 -7428.117} C_VEL
LIN {X 0,Y 473.809,Z 754.033,A -85,B 0,C 180,E1 -7429.258,E2 -7429.258} C_VEL
LIN {X 0,Y 473.901,Z 750.739,A -85,B 0,C 180,E1 -7430.459,E2 -7430.459} C_VEL
LIN {X 0,Y 474.038,Z 745.929,A -85,B 0,C 180,E1 -7431.792,E2 -7431.792} C_VEL
LIN {X 0,Y 474.243,Z 739.634,A -85,B 0,C 180,E1 -7433.154,E2 -7433.154} C_VEL
LIN {X 0,Y 474.6,Z 731.595,A -85,B 0,C 180,E1 -7434.534,E2 -7434.534} C_VEL
LIN {X 0,Y 475.041,Z 722.333,A -85,B 0,C 180,E1 -7435.792,E2 -7435.792} C_VEL
LIN {X 0,Y 475.46,Z 712.774,A -85,B 0,C 180,E1 -7436.844,E2 -7436.844} C_VEL
LIN {X 0,Y 475.977,Z 702.096,A -85,B 0,C 180,E1 -7437.795,E2 -7437.795} C_VEL
LIN {X 0,Y 476.414,Z 690.059,A -85,B 0,C 180,E1 -7438.636,E2 -7438.636} C_VEL
LIN {X 0,Y 476.885,Z 678.051,A -85,B 0,C 180,E1 -7439.279,E2 -7439.279} C_VEL
LIN {X 0,Y 476.946,Z 670.914,A -85,B 0,C 180,E1 -7439.584,E2 -7439.584} C_VEL
LIN {X 0,Y 475.92,Z 669.017,A -85,B 0,C 180,E1 -7439.687,E2 -7439.687} C_VEL
LIN {X 0,Y 469.266,Z 664.528,A -85,B 0,C 180,E1 -7440.061,E2 -7440.061} C_VEL
LIN {X 0,Y 468.426,Z 662.889,A -85,B 0,C 180,E1 -7440.139,E2 -7440.139} C_VEL
LIN {X 0,Y 466.738,Z 654.965,A -85,B 0,C 180,E1 -7440.429,E2 -7440.429} C_VEL
LIN {X 0,Y 466.829,Z 650.786,A -85,B 0,C 180,E1 -7443.151,E2 -7443.151} C_VEL
LIN {X 0,Y 466.937,Z 645.478,A -85,B 0,C 180,E1 -7446.655,E2 -7446.655} C_VEL
LIN {X 0,Y 467.049,Z 640.871,A -85,B 0,C 180,E1 -7449.751,E2 -7449.751} C_VEL
LIN {X 0,Y 467.165,Z 636.865,A -85,B 0,C 180,E1 -7452.489,E2 -7452.489} C_VEL
LIN {X 0,Y 467.3,Z 632.984,A -85,B 0,C 180,E1 -7455.186,E2 -7455.186} C_VEL
LIN {X 0,Y 467.479,Z 629.214,A -85,B 0,C 180,E1 -7457.85,E2 -7457.85} C_VEL
LIN {X 0,Y 467.451,Z 626.781,A -85,B 0,C 180,E1 -7459.606,E2 -7459.606} C_VEL
LIN {X 0,Y 467.54,Z 626.249,A -85,B 0,C 180,E1 -7460.482,E2 -7460.482} C_VEL
LIN {X 0,Y 467.713,Z 626.227,A -85,B 0,C 180,E1 -7463.095,E2 -7463.095} C_VEL
LIN {X 0,Y 467.727,Z 626.226,A -85,B 0,C 180,E1 -7464.827,E2 -7464.827} C_VEL
LIN {X 0,Y 467.863,Z 626.206,A -85,B 0,C 180,E1 -7467.417,E2 -7467.417} C_VEL
LIN {X 0,Y 467.887,Z 626.203,A -85,B 0,C 180,E1 -7470,E2 -7470} C_VEL
LIN {X 0,Y 467.863,Z 626.208,A -85,B 0,C 180,E1 -7472.582,E2 -7472.582} C_VEL
LIN {X 0,Y 467.736,Z 626.222,A -85,B 0,C 180,E1 -7476.037,E2 -7476.037} C_VEL
LIN {X 0,Y 467.583,Z 626.243,A -85,B 0,C 180,E1 -7478.644,E2 -7478.644} C_VEL
LIN {X 0,Y 467.216,Z 626.381,A -85,B 0,C 180,E1 -7481.371,E2 -7481.371} C_VEL
LIN {X 0,Y 467.074,Z 632.09,A -85,B 0,C 180,E1 -7484.82,E2 -7484.82} C_VEL
LIN {X 0,Y 466.957,Z 636.525,A -85,B 0,C 180,E1 -7487.518,E2 -7487.518} C_VEL
LIN {X 0,Y 466.888,Z 641.011,A -85,B 0,C 180,E1 -7490.255,E2 -7490.255} C_VEL
LIN {X 0,Y 466.822,Z 645.99,A -85,B 0,C 180,E1 -7493.313,E2 -7493.313} C_VEL
LIN {X 0,Y 466.751,Z 650.202,A -85,B 0,C 180,E1 -7495.89,E2 -7495.89} C_VEL
LIN {X 0,Y 466.733,Z 654.727,A -85,B 0,C 180,E1 -7498.683,E2 -7498.683} C_VEL
LIN {X 0,Y 469.602,Z 669.039,A -85,B 0,C 180,E1 -7499.211,E2 -7499.211} C_VEL
LIN {X 0,Y 470.108,Z 674.266,A -85,B 0,C 180,E1 -7499.437,E2 -7499.437} C_VEL
LIN {X 0,Y 469.645,Z 686.076,A -85,B 0,C 180,E1 -7500.019,E2 -7500.019} C_VEL
LIN {X 0,Y 469.216,Z 697.09,A -85,B 0,C 180,E1 -7500.727,E2 -7500.727} C_VEL
LIN {X 0,Y 468.724,Z 708.476,A -85,B 0,C 180,E1 -7501.653,E2 -7501.653} C_VEL
LIN {X 0,Y 468.21,Z 718.759,A -85,B 0,C 180,E1 -7502.708,E2 -7502.708} C_VEL
LIN {X 0,Y 467.757,Z 727.26,A -85,B 0,C 180,E1 -7503.774,E2 -7503.774} C_VEL
LIN {X 0,Y 467.364,Z 735.597,A -85,B 0,C 180,E1 -7505.054,E2 -7505.054} C_VEL
LIN {X 0,Y 467.084,Z 742.878,A -85,B 0,C 180,E1 -7506.465,E2 -7506.465} C_VEL
LIN {X 0,Y 466.92,Z 747.47,A -85,B 0,C 180,E1 -7507.566,E2 -7507.566} C_VEL
LIN {X 0,Y 466.768,Z 751.661,A -85,B 0,C 180,E1 -7508.821,E2 -7508.821} C_VEL
LIN {X 0,Y 466.583,Z 755.454,A -85,B 0,C 180,E1 -7510.367,E2 -7510.367} C_VEL
LIN {X 0,Y 466.541,Z 757.381,A -85,B 0,C 180,E1 -7511.514,E2 -7511.514} C_VEL
LIN {X 0,Y 466.522,Z 758.613,A -85,B 0,C 180,E1 -7512.68,E2 -7512.68} C_VEL
LIN {X 0,Y 466.528,Z 759.087,A -85,B 0,C 180,E1 -7513.864,E2 -7513.864} C_VEL
LIN {X 0,Y 466.564,Z 758.817,A -85,B 0,C 180,E1 -7515.07,E2 -7515.07} C_VEL
LIN {X 0,Y 466.529,Z 757.743,A -85,B 0,C 180,E1 -7516.31,E2 -7516.31} C_VEL
LIN {X 0,Y 466.659,Z 754.852,A -85,B 0,C 180,E1 -7518.037,E2 -7518.037} C_VEL
LIN {X 0,Y 466.788,Z 751.771,A -85,B 0,C 180,E1 -7519.248,E2 -7519.248} C_VEL
LIN {X 0,Y 466.97,Z 746.488,A -85,B 0,C 180,E1 -7520.794,E2 -7520.794} C_VEL
LIN {X 0,Y 467.176,Z 740.358,A -85,B 0,C 180,E1 -7522.165,E2 -7522.165} C_VEL
LIN {X 0,Y 467.545,Z 732.403,A -85,B 0,C 180,E1 -7523.576,E2 -7523.576} C_VEL
LIN {X 0,Y 467.981,Z 723.641,A -85,B 0,C 180,E1 -7524.809,E2 -7524.809} C_VEL
LIN {X 0,Y 468.461,Z 713.738,A -85,B 0,C 180,E1 -7525.938,E2 -7525.938} C_VEL
LIN {X 0,Y 469.008,Z 702.779,A -85,B 0,C 180,E1 -7526.937,E2 -7526.937} C_VEL
LIN {X 0,Y 469.48,Z 691.195,A -85,B 0,C 180,E1 -7527.771,E2 -7527.771} C_VEL
LIN {X 0,Y 470.006,Z 679.081,A -85,B 0,C 180,E1 -7528.442,E2 -7528.442} C_VEL
LIN {X 0,Y 469.999,Z 671.706,A -85,B 0,C 180,E1 -7528.766,E2 -7528.766} C_VEL
LIN {X 0,Y 467.88,Z 660.373,A -85,B 0,C 180,E1 -7529.22,E2 -7529.22} C_VEL
LIN {X 0,Y 466.75,Z 654.93,A -85,B 0,C 180,E1 -7529.41,E2 -7529.41} C_VEL
LIN {X 0,Y 466.789,Z 649.587,A -85,B 0,C 180,E1 -7532.66,E2 -7532.66} C_VEL
LIN {X 0,Y 466.826,Z 645.619,A -85,B 0,C 180,E1 -7535.068,E2 -7535.068} C_VEL
LIN {X 0,Y 466.883,Z 640.985,A -85,B 0,C 180,E1 -7537.894,E2 -7537.894} C_VEL
LIN {X 0,Y 466.963,Z 636.276,A -85,B 0,C 180,E1 -7540.664,E2 -7540.664} C_VEL
LIN {X 0,Y 467.006,Z 631.51,A -85,B 0,C 180,E1 -7543.385,E2 -7543.385} C_VEL
LIN {X 0,Y 467.085,Z 626.308,A -85,B 0,C 180,E1 -7546.347,E2 -7546.347} C_VEL
LIN {X 0,Y 467.511,Z 626.254,A -85,B 0,C 180,E1 -7548.73,E2 -7548.73} C_VEL
LIN {X 0,Y 467.676,Z 626.233,A -85,B 0,C 180,E1 -7551.357,E2 -7551.357} C_VEL
LIN {X 0,Y 467.741,Z 626.225,A -85,B 0,C 180,E1 -7553.963,E2 -7553.963} C_VEL
LIN {X 0,Y 467.858,Z 626.209,A -85,B 0,C 180,E1 -7557.417,E2 -7557.417} C_VEL
LIN {X 0,Y 467.879,Z 626.206,A -85,B 0,C 180,E1 -7560,E2 -7560} C_VEL
LIN {X 0,Y 467.857,Z 626.21,A -85,B 0,C 180,E1 -7562.583,E2 -7562.583} C_VEL
LIN {X 0,Y 467.741,Z 626.223,A -85,B 0,C 180,E1 -7566.037,E2 -7566.037} C_VEL
LIN {X 0,Y 467.679,Z 626.232,A -85,B 0,C 180,E1 -7568.643,E2 -7568.643} C_VEL
LIN {X 0,Y 467.653,Z 626.233,A -85,B 0,C 180,E1 -7572.146,E2 -7572.146} C_VEL
LIN {X 0,Y 467.635,Z 626.238,A -85,B 0,C 180,E1 -7575.695,E2 -7575.695} C_VEL
LIN {X 0,Y 467.614,Z 626.239,A -85,B 0,C 180,E1 -7578.765,E2 -7578.765} C_VEL
LIN {X 0,Y 467.577,Z 626.242,A -85,B 0,C 180,E1 -7581.269,E2 -7581.269} C_VEL
LIN {X 0,Y 467.57,Z 626.244,A -85,B 0,C 180,E1 -7583.943,E2 -7583.943} C_VEL
LIN {X 0,Y 467.624,Z 626.237,A -85,B 0,C 180,E1 -7586.8,E2 -7586.8} C_VEL
LIN {X 0,Y 467.585,Z 626.243,A -85,B 0,C 180,E1 -7589.736,E2 -7589.736} C_VEL
LIN {X 0,Y 467.581,Z 626.242,A -85,B 0,C 180,E1 -7592.759,E2 -7592.759} C_VEL
LIN {X 0,Y 467.553,Z 626.245,A -85,B 0,C 180,E1 -7595.89,E2 -7595.89} C_VEL
LIN {X 0,Y 467.58,Z 626.244,A -85,B 0,C 180,E1 -7599.145,E2 -7599.145} C_VEL
LIN {X 0,Y 467.584,Z 626.244,A -85,B 0,C 180,E1 -7602.567,E2 -7602.567} C_VEL
LIN {X 0,Y 467.568,Z 626.245,A -85,B 0,C 180,E1 -7605.054,E2 -7605.054} C_VEL
LIN {X 0,Y 467.587,Z 626.243,A -85,B 0,C 180,E1 -7607.44,E2 -7607.44} C_VEL
LIN {X 0,Y 467.62,Z 626.317,A -85,B 0,C 180,E1 -7610.86,E2 -7610.86} C_VEL
LIN {X 0,Y 468.343,Z 630.703,A -85,B 0,C 180,E1 -7613.113,E2 -7613.113} C_VEL
LIN {X 0,Y 468.566,Z 635.088,A -85,B 0,C 180,E1 -7615.253,E2 -7615.253} C_VEL
LIN {X 0,Y 468.222,Z 641.681,A -85,B 0,C 180,E1 -7618.309,E2 -7618.309} C_VEL
LIN {X 0,Y 468.017,Z 646.713,A -85,B 0,C 180,E1 -7620.571,E2 -7620.571} C_VEL
LIN {X 0,Y 467.688,Z 653.817,A -85,B 0,C 180,E1 -7623.686,E2 -7623.686} C_VEL
LIN {X 0,Y 467.477,Z 660.42,A -85,B 0,C 180,E1 -7626.501,E2 -7626.501} C_VEL
LIN {X 0,Y 467.268,Z 668.249,A -85,B 0,C 180,E1 -7629.762,E2 -7629.762} C_VEL
LIN {X 0,Y 467.064,Z 676.024,A -85,B 0,C 180,E1 -7632.938,E2 -7632.938} C_VEL
LIN {X 0,Y 467.006,Z 680.144,A -85,B 0,C 180,E1 -7634.598,E2 -7634.598} C_VEL
LIN {X 0,Y 469.322,Z 694.418,A -85,B 0,C 180,E1 -7635.077,E2 -7635.077} C_VEL
LIN {X 0,Y 470.009,Z 700.427,A -85,B 0,C 180,E1 -7635.33,E2 -7635.33} C_VEL
LIN {X 0,Y 469.578,Z 712.79,A -85,B 0,C 180,E1 -7635.925,E2 -7635.925} C_VEL
LIN {X 0,Y 469.129,Z 723.782,A -85,B 0,C 180,E1 -7636.618,E2 -7636.618} C_VEL
LIN {X 0,Y 468.669,Z 734.814,A -85,B 0,C 180,E1 -7637.499,E2 -7637.499} C_VEL
LIN {X 0,Y 468.157,Z 745.132,A -85,B 0,C 180,E1 -7638.527,E2 -7638.527} C_VEL
LIN {X 0,Y 467.678,Z 754.014,A -85,B 0,C 180,E1 -7639.612,E2 -7639.612} C_VEL
LIN {X 0,Y 467.302,Z 762.687,A -85,B 0,C 180,E1 -7640.915,E2 -7640.915} C_VEL
LIN {X 0,Y 467.016,Z 769.61,A -85,B 0,C 180,E1 -7642.216,E2 -7642.216} C_VEL
LIN {X 0,Y 466.814,Z 775.244,A -85,B 0,C 180,E1 -7643.54,E2 -7643.54} C_VEL
LIN {X 0,Y 466.772,Z 779.513,A -85,B 0,C 180,E1 -7644.817,E2 -7644.817} C_VEL
LIN {X 0,Y 466.659,Z 781.812,A -85,B 0,C 180,E1 -7645.682,E2 -7645.682} C_VEL
LIN {X 0,Y 466.693,Z 783.681,A -85,B 0,C 180,E1 -7646.547,E2 -7646.547} C_VEL
LIN {X 0,Y 466.646,Z 785.08,A -85,B 0,C 180,E1 -7647.411,E2 -7647.411} C_VEL
LIN {X 0,Y 466.618,Z 786.682,A -85,B 0,C 180,E1 -7649.137,E2 -7649.137} C_VEL
LIN {X 0,Y 466.598,Z 786.895,A -85,B 0,C 180,E1 -7650,E2 -7650} C_VEL
LIN {X 0,Y 466.618,Z 786.674,A -85,B 0,C 180,E1 -7650.863,E2 -7650.863} C_VEL
LIN {X 0,Y 466.646,Z 785.055,A -85,B 0,C 180,E1 -7652.59,E2 -7652.59} C_VEL
LIN {X 0,Y 466.693,Z 783.647,A -85,B 0,C 180,E1 -7653.454,E2 -7653.454} C_VEL
LIN {X 0,Y 466.701,Z 780.688,A -85,B 0,C 180,E1 -7654.751,E2 -7654.751} C_VEL
LIN {X 0,Y 466.794,Z 776.686,A -85,B 0,C 180,E1 -7656.05,E2 -7656.05} C_VEL
LIN {X 0,Y 466.981,Z 770.531,A -85,B 0,C 180,E1 -7657.567,E2 -7657.567} C_VEL
LIN {X 0,Y 467.258,Z 763.809,A -85,B 0,C 180,E1 -7658.869,E2 -7658.869} C_VEL
LIN {X 0,Y 467.609,Z 755.471,A -85,B 0,C 180,E1 -7660.172,E2 -7660.172} C_VEL
LIN {X 0,Y 468.026,Z 746.916,A -85,B 0,C 180,E1 -7661.257,E2 -7661.257} C_VEL
LIN {X 0,Y 468.589,Z 736.74,A -85,B 0,C 180,E1 -7662.305,E2 -7662.305} C_VEL
LIN {X 0,Y 468.951,Z 725.918,A -85,B 0,C 180,E1 -7663.212,E2 -7663.212} C_VEL
LIN {X 0,Y 469.45,Z 714.486,A -85,B 0,C 180,E1 -7663.97,E2 -7663.97} C_VEL
LIN {X 0,Y 469.908,Z 702.723,A -85,B 0,C 180,E1 -7664.564,E2 -7664.564} C_VEL
LIN {X 0,Y 469.74,Z 697.56,A -85,B 0,C 180,E1 -7664.785,E2 -7664.785} C_VEL
LIN {X 0,Y 467.677,Z 684.057,A -85,B 0,C 180,E1 -7665.275,E2 -7665.275} C_VEL
LIN {X 0,Y 466.974,Z 679.864,A -85,B 0,C 180,E1 -7665.398,E2 -7665.398} C_VEL
LIN {X 0,Y 467.124,Z 671.926,A -85,B 0,C 180,E1 -7668.585,E2 -7668.585} C_VEL
LIN {X 0,Y 467.353,Z 664.519,A -85,B 0,C 180,E1 -7671.619,E2 -7671.619} C_VEL
LIN {X 0,Y 467.551,Z 656.734,A -85,B 0,C 180,E1 -7674.891,E2 -7674.891} C_VEL
LIN {X 0,Y 467.834,Z 649.022,A -85,B 0,C 180,E1 -7678.243,E2 -7678.243} C_VEL
LIN {X 0,Y 468.128,Z 642.592,A -85,B 0,C 180,E1 -7681.158,E2 -7681.158} C_VEL
LIN {X 0,Y 468.437,Z 637.15,A -85,B 0,C 180,E1 -7683.719,E2 -7683.719} C_VEL
LIN {X 0,Y 468.541,Z 632.732,A -85,B 0,C 180,E1 -7685.905,E2 -7685.905} C_VEL
LIN {X 0,Y 467.833,Z 627.649,A -85,B 0,C 180,E1 -7688.632,E2 -7688.632} C_VEL
LIN {X 0,Y 467.614,Z 626.241,A -85,B 0,C 180,E1 -7689.49,E2 -7689.49} C_VEL
LIN {X 0,Y 467.589,Z 626.244,A -85,B 0,C 180,E1 -7692.567,E2 -7692.567} C_VEL
LIN {X 0,Y 467.573,Z 626.245,A -85,B 0,C 180,E1 -7695.053,E2 -7695.053} C_VEL
LIN {X 0,Y 467.591,Z 626.244,A -85,B 0,C 180,E1 -7697.44,E2 -7697.44} C_VEL
LIN {X 0,Y 467.584,Z 626.244,A -85,B 0,C 180,E1 -7700.855,E2 -7700.855} C_VEL
LIN {X 0,Y 467.562,Z 626.247,A -85,B 0,C 180,E1 -7704.261,E2 -7704.261} C_VEL
LIN {X 0,Y 467.584,Z 626.244,A -85,B 0,C 180,E1 -7707.321,E2 -7707.321} C_VEL
LIN {X 0,Y 467.572,Z 626.245,A -85,B 0,C 180,E1 -7710.667,E2 -7710.667} C_VEL
LIN {X 0,Y 467.618,Z 626.239,A -85,B 0,C 180,E1 -7713.2,E2 -7713.2} C_VEL
LIN {X 0,Y 467.594,Z 626.241,A -85,B 0,C 180,E1 -7716.468,E2 -7716.468} C_VEL
LIN {X 0,Y 467.626,Z 626.238,A -85,B 0,C 180,E1 -7719.777,E2 -7719.777} C_VEL
LIN {X 0,Y 467.611,Z 626.241,A -85,B 0,C 180,E1 -7722.507,E2 -7722.507} C_VEL
LIN {X 0,Y 467.608,Z 626.239,A -85,B 0,C 180,E1 -7725.196,E2 -7725.196} C_VEL
LIN {X 0,Y 467.657,Z 626.234,A -85,B 0,C 180,E1 -7727.855,E2 -7727.855} C_VEL
LIN {X 0,Y 467.684,Z 626.231,A -85,B 0,C 180,E1 -7731.357,E2 -7731.357} C_VEL
LIN {X 0,Y 467.745,Z 626.222,A -85,B 0,C 180,E1 -7733.963,E2 -7733.963} C_VEL
LIN {X 0,Y 467.861,Z 626.208,A -85,B 0,C 180,E1 -7737.417,E2 -7737.417} C_VEL
LIN {X 0,Y 467.884,Z 626.206,A -85,B 0,C 180,E1 -7740,E2 -7740} C_VEL
LIN {X 0,Y 467.862,Z 626.21,A -85,B 0,C 180,E1 -7742.583,E2 -7742.583} C_VEL
LIN {X 0,Y 467.746,Z 626.224,A -85,B 0,C 180,E1 -7746.037,E2 -7746.037} C_VEL
LIN {X 0,Y 467.661,Z 626.235,A -85,B 0,C 180,E1 -7748.643,E2 -7748.643} C_VEL
LIN {X 0,Y 467.6,Z 626.475,A -85,B 0,C 180,E1 -7749.516,E2 -7749.516} C_VEL
LIN {X 0,Y 467.518,Z 630.148,A -85,B 0,C 180,E1 -7752.281,E2 -7752.281} C_VEL
LIN {X 0,Y 467.34,Z 634.921,A -85,B 0,C 180,E1 -7755.751,E2 -7755.751} C_VEL
LIN {X 0,Y 467.167,Z 639.957,A -85,B 0,C 180,E1 -7759.327,E2 -7759.327} C_VEL
LIN {X 0,Y 467.032,Z 643.992,A -85,B 0,C 180,E1 -7762.099,E2 -7762.099} C_VEL
LIN {X 0,Y 466.942,Z 648.904,A -85,B 0,C 180,E1 -7765.436,E2 -7765.436} C_VEL
LIN {X 0,Y 466.815,Z 652.492,A -85,B 0,C 180,E1 -7767.821,E2 -7767.821} C_VEL
LIN {X 0,Y 466.752,Z 655.308,A -85,B 0,C 180,E1 -7769.673,E2 -7769.673} C_VEL
LIN {X 0,Y 469.71,Z 669.383,A -85,B 0,C 180,E1 -7770.206,E2 -7770.206} C_VEL
LIN {X 0,Y 470.109,Z 674.499,A -85,B 0,C 180,E1 -7770.426,E2 -7770.426} C_VEL
LIN {X 0,Y 469.699,Z 686.471,A -85,B 0,C 180,E1 -7771.016,E2 -7771.016} C_VEL
LIN {X 0,Y 469.236,Z 697.702,A -85,B 0,C 180,E1 -7771.742,E2 -7771.742} C_VEL
LIN {X 0,Y 468.705,Z 708.951,A -85,B 0,C 180,E1 -7772.67,E2 -7772.67} C_VEL
LIN {X 0,Y 468.22,Z 719.301,A -85,B 0,C 180,E1 -7773.736,E2 -7773.736} C_VEL
LIN {X 0,Y 467.829,Z 727.787,A -85,B 0,C 180,E1 -7774.81,E2 -7774.81} C_VEL
LIN {X 0,Y 467.39,Z 736.452,A -85,B 0,C 180,E1 -7776.171,E2 -7776.171} C_VEL
LIN {X 0,Y 467.087,Z 743.574,A -85,B 0,C 180,E1 -7777.576,E2 -7777.576} C_VEL
LIN {X 0,Y 466.873,Z 748.581,A -85,B 0,C 180,E1 -7778.825,E2 -7778.825} C_VEL
LIN {X 0,Y 466.755,Z 753.263,A -85,B 0,C 180,E1 -7780.35,E2 -7780.35} C_VEL
LIN {X 0,Y 466.67,Z 755.849,A -85,B 0,C 180,E1 -7781.501,E2 -7781.501} C_VEL
LIN {X 0,Y 466.561,Z 757.694,A -85,B 0,C 180,E1 -7782.676,E2 -7782.676} C_VEL
LIN {X 0,Y 466.533,Z 758.813,A -85,B 0,C 180,E1 -7783.865,E2 -7783.865} C_VEL
LIN {X 0,Y 466.567,Z 759.193,A -85,B 0,C 180,E1 -7785.07,E2 -7785.07} C_VEL
LIN {X 0,Y 466.527,Z 758.75,A -85,B 0,C 180,E1 -7786.311,E2 -7786.311} C_VEL
LIN {X 0,Y 466.569,Z 757.462,A -85,B 0,C 180,E1 -7787.57,E2 -7787.57} C_VEL
LIN {X 0,Y 466.694,Z 755.273,A -85,B 0,C 180,E1 -7788.847,E2 -7788.847} C_VEL
LIN {X 0,Y 466.801,Z 752.045,A -85,B 0,C 180,E1 -7790.16,E2 -7790.16} C_VEL
LIN {X 0,Y 466.931,Z 747.614,A -85,B 0,C 180,E1 -7791.507,E2 -7791.507} C_VEL
LIN {X 0,Y 467.168,Z 741.21,A -85,B 0,C 180,E1 -7793.004,E2 -7793.004} C_VEL
LIN {X 0,Y 467.514,Z 734.312,A -85,B 0,C 180,E1 -7794.269,E2 -7794.269} C_VEL
LIN {X 0,Y 467.876,Z 726.23,A -85,B 0,C 180,E1 -7795.473,E2 -7795.473} C_VEL
LIN {X 0,Y 468.327,Z 716.817,A -85,B 0,C 180,E1 -7796.616,E2 -7796.616} C_VEL
LIN {X 0,Y 468.812,Z 706.923,A -85,B 0,C 180,E1 -7797.593,E2 -7797.593} C_VEL
LIN {X 0,Y 469.282,Z 695.966,A -85,B 0,C 180,E1 -7798.459,E2 -7798.459} C_VEL
LIN {X 0,Y 469.783,Z 683.284,A -85,B 0,C 180,E1 -7799.239,E2 -7799.239} C_VEL
LIN {X 0,Y 470.097,Z 672.098,A -85,B 0,C 180,E1 -7799.759,E2 -7799.759} C_VEL
LIN {X 0,Y 468.426,Z 662.889,A -85,B 0,C 180,E1 -7800.139,E2 -7800.139} C_VEL
LIN {X 0,Y 467.468,Z 659.678,A -85,B 0,C 180,E1 -7800.347,E2 -7800.347} C_VEL
LIN {X 0,Y 466.169,Z 657.177,A -85,B 0,C 180,E1 -7800.661,E2 -7800.661} C_VEL
LIN {X 0,Y 464.006,Z 654.558,A -85,B 0,C 180,E1 -7801.252,E2 -7801.252} C_VEL
LIN {X 0,Y 461.931,Z 653.031,A -85,B 0,C 180,E1 -7801.952,E2 -7801.952} C_VEL
LIN {X 0,Y 460.016,Z 651.64,A -85,B 0,C 180,E1 -7802.968,E2 -7802.968} C_VEL
LIN {X 0,Y 459.753,Z 650.875,A -85,B 0,C 180,E1 -7803.488,E2 -7803.488} C_VEL
LIN {X 0,Y 459.864,Z 646.237,A -85,B 0,C 180,E1 -7806.587,E2 -7806.587} C_VEL
LIN {X 0,Y 459.992,Z 642.056,A -85,B 0,C 180,E1 -7809.426,E2 -7809.426} C_VEL
LIN {X 0,Y 460.093,Z 638.019,A -85,B 0,C 180,E1 -7812.211,E2 -7812.211} C_VEL
LIN {X 0,Y 460.229,Z 634.114,A -85,B 0,C 180,E1 -7814.953,E2 -7814.953} C_VEL
LIN {X 0,Y 460.398,Z 630.286,A -85,B 0,C 180,E1 -7817.679,E2 -7817.679} C_VEL
LIN {X 0,Y 460.403,Z 627.872,A -85,B 0,C 180,E1 -7819.445,E2 -7819.445} C_VEL
LIN {X 0,Y 460.472,Z 627.129,A -85,B 0,C 180,E1 -7820.335,E2 -7820.335} C_VEL
LIN {X 0,Y 460.674,Z 627.104,A -85,B 0,C 180,E1 -7822.989,E2 -7822.989} C_VEL
LIN {X 0,Y 460.7,Z 627.101,A -85,B 0,C 180,E1 -7824.748,E2 -7824.748} C_VEL
LIN {X 0,Y 460.828,Z 627.083,A -85,B 0,C 180,E1 -7827.377,E2 -7827.377} C_VEL
LIN {X 0,Y 460.858,Z 627.078,A -85,B 0,C 180,E1 -7830,E2 -7830} C_VEL
LIN {X 0,Y 460.828,Z 627.084,A -85,B 0,C 180,E1 -7832.622,E2 -7832.622} C_VEL
LIN {X 0,Y 460.701,Z 627.098,A -85,B 0,C 180,E1 -7836.13,E2 -7836.13} C_VEL
LIN {X 0,Y 460.536,Z 627.121,A -85,B 0,C 180,E1 -7838.777,E2 -7838.777} C_VEL
LIN {X 0,Y 460.146,Z 627.252,A -85,B 0,C 180,E1 -7841.452,E2 -7841.452} C_VEL
LIN {X 0,Y 460.019,Z 633.154,A -85,B 0,C 180,E1 -7845.053,E2 -7845.053} C_VEL
LIN {X 0,Y 459.883,Z 639.013,A -85,B 0,C 180,E1 -7848.649,E2 -7848.649} C_VEL
LIN {X 0,Y 459.78,Z 643.687,A -85,B 0,C 180,E1 -7851.521,E2 -7851.521} C_VEL
LIN {X 0,Y 459.695,Z 648.31,A -85,B 0,C 180,E1 -7854.379,E2 -7854.379} C_VEL
LIN {X 0,Y 459.645,Z 653.395,A -85,B 0,C 180,E1 -7857.523,E2 -7857.523} C_VEL
LIN {X 0,Y 459.632,Z 654.891,A -85,B 0,C 180,E1 -7858.45,E2 -7858.45} C_VEL
LIN {X 0,Y 462.617,Z 669.359,A -85,B 0,C 180,E1 -7858.993,E2 -7858.993} C_VEL
LIN {X 0,Y 463.248,Z 674.243,A -85,B 0,C 180,E1 -7859.212,E2 -7859.212} C_VEL
LIN {X 0,Y 462.726,Z 686.946,A -85,B 0,C 180,E1 -7859.852,E2 -7859.852} C_VEL
LIN {X 0,Y 462.264,Z 698.476,A -85,B 0,C 180,E1 -7860.618,E2 -7860.618} C_VEL
LIN {X 0,Y 461.74,Z 709.292,A -85,B 0,C 180,E1 -7861.53,E2 -7861.53} C_VEL
LIN {X 0,Y 461.211,Z 719.617,A -85,B 0,C 180,E1 -7862.618,E2 -7862.618} C_VEL
LIN {X 0,Y 460.68,Z 728.988,A -85,B 0,C 180,E1 -7863.836,E2 -7863.836} C_VEL
LIN {X 0,Y 460.272,Z 737.383,A -85,B 0,C 180,E1 -7865.209,E2 -7865.209} C_VEL
LIN {X 0,Y 459.986,Z 744.064,A -85,B 0,C 180,E1 -7866.574,E2 -7866.574} C_VEL
LIN {X 0,Y 459.815,Z 748.447,A -85,B 0,C 180,E1 -7867.688,E2 -7867.688} C_VEL
LIN {X 0,Y 459.69,Z 752.052,A -85,B 0,C 180,E1 -7868.816,E2 -7868.816} C_VEL
LIN {X 0,Y 459.521,Z 755.255,A -85,B 0,C 180,E1 -7870.119,E2 -7870.119} C_VEL
LIN {X 0,Y 459.446,Z 757.538,A -85,B 0,C 180,E1 -7871.449,E2 -7871.449} C_VEL
LIN {X 0,Y 459.433,Z 758.865,A -85,B 0,C 180,E1 -7872.755,E2 -7872.755} C_VEL
LIN {X 0,Y 459.441,Z 759.311,A -85,B 0,C 180,E1 -7874.032,E2 -7874.032} C_VEL
LIN {X 0,Y 459.462,Z 758.909,A -85,B 0,C 180,E1 -7875.281,E2 -7875.281} C_VEL
LIN {X 0,Y 459.46,Z 757.74,A -85,B 0,C 180,E1 -7876.502,E2 -7876.502} C_VEL
LIN {X 0,Y 459.515,Z 755.829,A -85,B 0,C 180,E1 -7877.704,E2 -7877.704} C_VEL
LIN {X 0,Y 459.673,Z 753.155,A -85,B 0,C 180,E1 -7878.895,E2 -7878.895} C_VEL
LIN {X 0,Y 459.814,Z 748.713,A -85,B 0,C 180,E1 -7880.348,E2 -7880.348} C_VEL
LIN {X 0,Y 460.045,Z 742.976,A -85,B 0,C 180,E1 -7881.778,E2 -7881.778} C_VEL
LIN {X 0,Y 460.324,Z 736.712,A -85,B 0,C 180,E1 -7883.022,E2 -7883.022} C_VEL
LIN {X 0,Y 460.719,Z 728.977,A -85,B 0,C 180,E1 -7884.274,E2 -7884.274} C_VEL
LIN {X 0,Y 461.163,Z 720.573,A -85,B 0,C 180,E1 -7885.38,E2 -7885.38} C_VEL
LIN {X 0,Y 461.714,Z 709.978,A -85,B 0,C 180,E1 -7886.51,E2 -7886.51} C_VEL
LIN {X 0,Y 462.252,Z 698.801,A -85,B 0,C 180,E1 -7887.463,E2 -7887.463} C_VEL
LIN {X 0,Y 462.784,Z 686.808,A -85,B 0,C 180,E1 -7888.258,E2 -7888.258} C_VEL
LIN {X 0,Y 463.269,Z 674.781,A -85,B 0,C 180,E1 -7888.864,E2 -7888.864} C_VEL
LIN {X 0,Y 461.718,Z 664.487,A -85,B 0,C 180,E1 -7889.31,E2 -7889.31} C_VEL
LIN {X 0,Y 459.657,Z 655.117,A -85,B 0,C 180,E1 -7889.65,E2 -7889.65} C_VEL
LIN {X 0,Y 459.729,Z 650.149,A -85,B 0,C 180,E1 -7892.702,E2 -7892.702} C_VEL
LIN {X 0,Y 459.779,Z 645.327,A -85,B 0,C 180,E1 -7895.625,E2 -7895.625} C_VEL
LIN {X 0,Y 459.847,Z 640.084,A -85,B 0,C 180,E1 -7898.792,E2 -7898.792} C_VEL
LIN {X 0,Y 459.945,Z 635.795,A -85,B 0,C 180,E1 -7901.326,E2 -7901.326} C_VEL
LIN {X 0,Y 460.025,Z 629.508,A -85,B 0,C 180,E1 -7904.947,E2 -7904.947} C_VEL
LIN {X 0,Y 460.028,Z 627.188,A -85,B 0,C 180,E1 -7906.302,E2 -7906.302} C_VEL
LIN {X 0,Y 460.446,Z 627.134,A -85,B 0,C 180,E1 -7908.555,E2 -7908.555} C_VEL
LIN {X 0,Y 460.621,Z 627.112,A -85,B 0,C 180,E1 -7911.224,E2 -7911.224} C_VEL
LIN {X 0,Y 460.706,Z 627.101,A -85,B 0,C 180,E1 -7913.87,E2 -7913.87} C_VEL
LIN {X 0,Y 460.823,Z 627.086,A -85,B 0,C 180,E1 -7917.378,E2 -7917.378} C_VEL
LIN {X 0,Y 460.85,Z 627.082,A -85,B 0,C 180,E1 -7920,E2 -7920} C_VEL
LIN {X 0,Y 460.822,Z 627.086,A -85,B 0,C 180,E1 -7922.622,E2 -7922.622} C_VEL
LIN {X 0,Y 460.707,Z 627.099,A -85,B 0,C 180,E1 -7926.13,E2 -7926.13} C_VEL
LIN {X 0,Y 460.626,Z 627.11,A -85,B 0,C 180,E1 -7928.776,E2 -7928.776} C_VEL
LIN {X 0,Y 460.609,Z 627.111,A -85,B 0,C 180,E1 -7932.445,E2 -7932.445} C_VEL
LIN {X 0,Y 460.596,Z 627.113,A -85,B 0,C 180,E1 -7935.998,E2 -7935.998} C_VEL
LIN {X 0,Y 460.567,Z 627.116,A -85,B 0,C 180,E1 -7938.902,E2 -7938.902} C_VEL
LIN {X 0,Y 460.512,Z 627.121,A -85,B 0,C 180,E1 -7941.486,E2 -7941.486} C_VEL
LIN {X 0,Y 460.539,Z 627.12,A -85,B 0,C 180,E1 -7944.332,E2 -7944.332} C_VEL
LIN {X 0,Y 460.581,Z 627.116,A -85,B 0,C 180,E1 -7947.243,E2 -7947.243} C_VEL
LIN {X 0,Y 460.524,Z 627.122,A -85,B 0,C 180,E1 -7950.239,E2 -7950.239} C_VEL
LIN {X 0,Y 460.526,Z 627.122,A -85,B 0,C 180,E1 -7953.325,E2 -7953.325} C_VEL
LIN {X 0,Y 460.475,Z 627.129,A -85,B 0,C 180,E1 -7956.53,E2 -7956.53} C_VEL
LIN {X 0,Y 460.542,Z 627.12,A -85,B 0,C 180,E1 -7958.898,E2 -7958.898} C_VEL
LIN {X 0,Y 460.52,Z 627.121,A -85,B 0,C 180,E1 -7962.182,E2 -7962.182} C_VEL
LIN {X 0,Y 460.515,Z 627.124,A -85,B 0,C 180,E1 -7965.412,E2 -7965.412} C_VEL
LIN {X 0,Y 460.53,Z 627.122,A -85,B 0,C 180,E1 -7968.398,E2 -7968.398} C_VEL
LIN {X 0,Y 460.565,Z 627.173,A -85,B 0,C 180,E1 -7970.647,E2 -7970.647} C_VEL
LIN {X 0,Y 461.432,Z 632.787,A -85,B 0,C 180,E1 -7973.559,E2 -7973.559} C_VEL
LIN {X 0,Y 461.537,Z 636.363,A -85,B 0,C 180,E1 -7975.314,E2 -7975.314} C_VEL
LIN {X 0,Y 461.148,Z 643.758,A -85,B 0,C 180,E1 -7978.791,E2 -7978.791} C_VEL
LIN {X 0,Y 460.864,Z 650.375,A -85,B 0,C 180,E1 -7981.788,E2 -7981.788} C_VEL
LIN {X 0,Y 460.53,Z 658.11,A -85,B 0,C 180,E1 -7985.187,E2 -7985.187} C_VEL
LIN {X 0,Y 460.277,Z 665.866,A -85,B 0,C 180,E1 -7988.503,E2 -7988.503} C_VEL
LIN {X 0,Y 460.048,Z 673.624,A -85,B 0,C 180,E1 -7991.75,E2 -7991.75} C_VEL
LIN {X 0,Y 459.917,Z 680.006,A -85,B 0,C 180,E1 -7994.371,E2 -7994.371} C_VEL
LIN {X 0,Y 462.166,Z 693.834,A -85,B 0,C 180,E1 -7994.83,E2 -7994.83} C_VEL
LIN {X 0,Y 463.085,Z 701.437,A -85,B 0,C 180,E1 -7995.162,E2 -7995.162} C_VEL
LIN {X 0,Y 462.676,Z 712.525,A -85,B 0,C 180,E1 -7995.71,E2 -7995.71} C_VEL
LIN {X 0,Y 462.169,Z 724.462,A -85,B 0,C 180,E1 -7996.48,E2 -7996.48} C_VEL
LIN {X 0,Y 461.678,Z 735.027,A -85,B 0,C 180,E1 -7997.349,E2 -7997.349} C_VEL
LIN {X 0,Y 461.152,Z 744.899,A -85,B 0,C 180,E1 -7998.351,E2 -7998.351} C_VEL
LIN {X 0,Y 460.658,Z 753.786,A -85,B 0,C 180,E1 -7999.451,E2 -7999.451} C_VEL
LIN {X 0,Y 460.263,Z 762.465,A -85,B 0,C 180,E1 -8000.774,E2 -8000.774} C_VEL
LIN {X 0,Y 459.955,Z 769.392,A -85,B 0,C 180,E1 -8002.096,E2 -8002.096} C_VEL
LIN {X 0,Y 459.72,Z 775.481,A -85,B 0,C 180,E1 -8003.562,E2 -8003.562} C_VEL
LIN {X 0,Y 459.631,Z 780.53,A -85,B 0,C 180,E1 -8005.176,E2 -8005.176} C_VEL
LIN {X 0,Y 459.589,Z 783.47,A -85,B 0,C 180,E1 -8006.494,E2 -8006.494} C_VEL
LIN {X 0,Y 459.57,Z 784.87,A -85,B 0,C 180,E1 -8007.371,E2 -8007.371} C_VEL
LIN {X 0,Y 459.521,Z 786.472,A -85,B 0,C 180,E1 -8009.124,E2 -8009.124} C_VEL
LIN {X 0,Y 459.53,Z 786.685,A -85,B 0,C 180,E1 -8010,E2 -8010} C_VEL
LIN {X 0,Y 459.521,Z 786.462,A -85,B 0,C 180,E1 -8010.877,E2 -8010.877} C_VEL
LIN {X 0,Y 459.57,Z 784.84,A -85,B 0,C 180,E1 -8012.63,E2 -8012.63} C_VEL
LIN {X 0,Y 459.589,Z 783.429,A -85,B 0,C 180,E1 -8013.507,E2 -8013.507} C_VEL
LIN {X 0,Y 459.631,Z 780.468,A -85,B 0,C 180,E1 -8014.824,E2 -8014.824} C_VEL
LIN {X 0,Y 459.718,Z 776.46,A -85,B 0,C 180,E1 -8016.144,E2 -8016.144} C_VEL
LIN {X 0,Y 459.911,Z 770.296,A -85,B 0,C 180,E1 -8017.684,E2 -8017.684} C_VEL
LIN {X 0,Y 460.188,Z 763.569,A -85,B 0,C 180,E1 -8019.006,E2 -8019.006} C_VEL
LIN {X 0,Y 460.566,Z 755.229,A -85,B 0,C 180,E1 -8020.329,E2 -8020.329} C_VEL
LIN {X 0,Y 461.021,Z 746.672,A -85,B 0,C 180,E1 -8021.431,E2 -8021.431} C_VEL
LIN {X 0,Y 461.603,Z 736.713,A -85,B 0,C 180,E1 -8022.474,E2 -8022.474} C_VEL
LIN {X 0,Y 462.023,Z 725.678,A -85,B 0,C 180,E1 -8023.414,E2 -8023.414} C_VEL
LIN {X 0,Y 462.554,Z 714.247,A -85,B 0,C 180,E1 -8024.182,E2 -8024.182} C_VEL
LIN {X 0,Y 463.043,Z 702.49,A -85,B 0,C 180,E1 -8024.784,E2 -8024.784} C_VEL
LIN {X 0,Y 462.871,Z 698.615,A -85,B 0,C 180,E1 -8024.959,E2 -8024.959} C_VEL
LIN {X 0,Y 460.82,Z 685.074,A -85,B 0,C 180,E1 -8025.477,E2 -8025.477} C_VEL
LIN {X 0,Y 459.897,Z 679.638,A -85,B 0,C 180,E1 -8025.649,E2 -8025.649} C_VEL
LIN {X 0,Y 460.054,Z 672.148,A -85,B 0,C 180,E1 -8028.712,E2 -8028.712} C_VEL
LIN {X 0,Y 460.273,Z 665.458,A -85,B 0,C 180,E1 -8031.498,E2 -8031.498} C_VEL
LIN {X 0,Y 460.535,Z 656.589,A -85,B 0,C 180,E1 -8035.296,E2 -8035.296} C_VEL
LIN {X 0,Y 460.873,Z 648.919,A -85,B 0,C 180,E1 -8038.709,E2 -8038.709} C_VEL
LIN {X 0,Y 461.146,Z 643.096,A -85,B 0,C 180,E1 -8041.41,E2 -8041.41} C_VEL
LIN {X 0,Y 461.522,Z 636.342,A -85,B 0,C 180,E1 -8044.684,E2 -8044.684} C_VEL
LIN {X 0,Y 461.336,Z 631.898,A -85,B 0,C 180,E1 -8046.995,E2 -8046.995} C_VEL
LIN {X 0,Y 460.558,Z 627.12,A -85,B 0,C 180,E1 -8049.735,E2 -8049.735} C_VEL
LIN {X 0,Y 460.519,Z 627.125,A -85,B 0,C 180,E1 -8052.901,E2 -8052.901} C_VEL
LIN {X 0,Y 460.513,Z 627.123,A -85,B 0,C 180,E1 -8055.83,E2 -8055.83} C_VEL
LIN {X 0,Y 460.533,Z 627.123,A -85,B 0,C 180,E1 -8058.989,E2 -8058.989} C_VEL
LIN {X 0,Y 460.528,Z 627.124,A -85,B 0,C 180,E1 -8061.267,E2 -8061.267} C_VEL
LIN {X 0,Y 460.513,Z 627.124,A -85,B 0,C 180,E1 -8064.554,E2 -8064.554} C_VEL
LIN {X 0,Y 460.533,Z 627.12,A -85,B 0,C 180,E1 -8067.716,E2 -8067.716} C_VEL
LIN {X 0,Y 460.542,Z 627.12,A -85,B 0,C 180,E1 -8070.769,E2 -8070.769} C_VEL
LIN {X 0,Y 460.565,Z 627.116,A -85,B 0,C 180,E1 -8073.735,E2 -8073.735} C_VEL
LIN {X 0,Y 460.548,Z 627.12,A -85,B 0,C 180,E1 -8076.624,E2 -8076.624} C_VEL
LIN {X 0,Y 460.554,Z 627.119,A -85,B 0,C 180,E1 -8079.453,E2 -8079.453} C_VEL
LIN {X 0,Y 460.561,Z 627.118,A -85,B 0,C 180,E1 -8082.23,E2 -8082.23} C_VEL
LIN {X 0,Y 460.567,Z 627.117,A -85,B 0,C 180,E1 -8084.965,E2 -8084.965} C_VEL
LIN {X 0,Y 460.613,Z 627.112,A -85,B 0,C 180,E1 -8088.559,E2 -8088.559} C_VEL
LIN {X 0,Y 460.697,Z 627.099,A -85,B 0,C 180,E1 -8092.109,E2 -8092.109} C_VEL
LIN {X 0,Y 460.698,Z 627.102,A -85,B 0,C 180,E1 -8094.748,E2 -8094.748} C_VEL
LIN {X 0,Y 460.802,Z 627.087,A -85,B 0,C 180,E1 -8097.378,E2 -8097.378} C_VEL
LIN {X 0,Y 460.855,Z 627.081,A -85,B 0,C 180,E1 -8100,E2 -8100} C_VEL
LIN {X 0,Y 460.827,Z 627.087,A -85,B 0,C 180,E1 -8102.622,E2 -8102.622} C_VEL
LIN {X 0,Y 460.712,Z 627.099,A -85,B 0,C 180,E1 -8106.13,E2 -8106.13} C_VEL
LIN {X 0,Y 460.605,Z 627.114,A -85,B 0,C 180,E1 -8108.777,E2 -8108.777} C_VEL
LIN {X 0,Y 460.561,Z 627.663,A -85,B 0,C 180,E1 -8109.663,E2 -8109.663} C_VEL
LIN {X 0,Y 460.466,Z 631.207,A -85,B 0,C 180,E1 -8112.361,E2 -8112.361} C_VEL
LIN {X 0,Y 460.261,Z 636.058,A -85,B 0,C 180,E1 -8115.953,E2 -8115.953} C_VEL
LIN {X 0,Y 460.167,Z 639.957,A -85,B 0,C 180,E1 -8118.754,E2 -8118.754} C_VEL
LIN {X 0,Y 459.996,Z 643.881,A -85,B 0,C 180,E1 -8121.511,E2 -8121.511} C_VEL
LIN {X 0,Y 459.873,Z 648.018,A -85,B 0,C 180,E1 -8124.37,E2 -8124.37} C_VEL
LIN {X 0,Y 459.83,Z 652.331,A -85,B 0,C 180,E1 -8127.292,E2 -8127.292} C_VEL
LIN {X 0,Y 459.729,Z 655.681,A -85,B 0,C 180,E1 -8129.445,E2 -8129.445} C_VEL
LIN {X 0,Y 462.558,Z 668.715,A -85,B 0,C 180,E1 -8129.937,E2 -8129.937} C_VEL
LIN {X 0,Y 463.258,Z 674.379,A -85,B 0,C 180,E1 -8130.19,E2 -8130.19} C_VEL
LIN {X 0,Y 462.842,Z 686.671,A -85,B 0,C 180,E1 -8130.804,E2 -8130.804} C_VEL
LIN {X 0,Y 462.359,Z 697.282,A -85,B 0,C 180,E1 -8131.493,E2 -8131.493} C_VEL
LIN {X 0,Y 461.822,Z 708.725,A -85,B 0,C 180,E1 -8132.441,E2 -8132.441} C_VEL
LIN {X 0,Y 461.256,Z 719.196,A -85,B 0,C 180,E1 -8133.527,E2 -8133.527} C_VEL
LIN {X 0,Y 460.81,Z 728.512,A -85,B 0,C 180,E1 -8134.727,E2 -8134.727} C_VEL
LIN {X 0,Y 460.393,Z 736.447,A -85,B 0,C 180,E1 -8135.996,E2 -8135.996} C_VEL
LIN {X 0,Y 460.046,Z 743.514,A -85,B 0,C 180,E1 -8137.402,E2 -8137.402} C_VEL
LIN {X 0,Y 459.806,Z 749.068,A -85,B 0,C 180,E1 -8138.805,E2 -8138.805} C_VEL
LIN {X 0,Y 459.681,Z 753.131,A -85,B 0,C 180,E1 -8140.142,E2 -8140.142} C_VEL
LIN {X 0,Y 459.579,Z 756.104,A -85,B 0,C 180,E1 -8141.468,E2 -8141.468} C_VEL
LIN {X 0,Y 459.467,Z 758.057,A -85,B 0,C 180,E1 -8142.76,E2 -8142.76} C_VEL
LIN {X 0,Y 459.445,Z 759.123,A -85,B 0,C 180,E1 -8144.032,E2 -8144.032} C_VEL
LIN {X 0,Y 459.465,Z 759.367,A -85,B 0,C 180,E1 -8145.282,E2 -8145.282} C_VEL
LIN {X 0,Y 459.436,Z 758.85,A -85,B 0,C 180,E1 -8146.499,E2 -8146.499} C_VEL
LIN {X 0,Y 459.482,Z 757.55,A -85,B 0,C 180,E1 -8147.701,E2 -8147.701} C_VEL
LIN {X 0,Y 459.603,Z 755.513,A -85,B 0,C 180,E1 -8148.888,E2 -8148.888} C_VEL
LIN {X 0,Y 459.701,Z 752.777,A -85,B 0,C 180,E1 -8150.051,E2 -8150.051} C_VEL
LIN {X 0,Y 459.849,Z 748.215,A -85,B 0,C 180,E1 -8151.495,E2 -8151.495} C_VEL
LIN {X 0,Y 460.099,Z 741.877,A -85,B 0,C 180,E1 -8153.024,E2 -8153.024} C_VEL
LIN {X 0,Y 460.439,Z 735.233,A -85,B 0,C 180,E1 -8154.288,E2 -8154.288} C_VEL
LIN {X 0,Y 460.9,Z 726.25,A -85,B 0,C 180,E1 -8155.654,E2 -8155.654} C_VEL
LIN {X 0,Y 461.417,Z 716.022,A -85,B 0,C 180,E1 -8156.901,E2 -8156.901} C_VEL
LIN {X 0,Y 461.904,Z 706.629,A -85,B 0,C 180,E1 -8157.823,E2 -8157.823} C_VEL
LIN {X 0,Y 462.412,Z 695.527,A -85,B 0,C 180,E1 -8158.702,E2 -8158.702} C_VEL
LIN {X 0,Y 462.938,Z 682.911,A -85,B 0,C 180,E1 -8159.481,E2 -8159.481} C_VEL
LIN {X 0,Y 463.202,Z 672.867,A -85,B 0,C 180,E1 -8159.954,E2 -8159.954} C_VEL
LIN {X 0,Y 460.931,Z 661.036,A -85,B 0,C 180,E1 -8160.45,E2 -8160.45} C_VEL
LIN {X 0,Y 459.67,Z 655.194,A -85,B 0,C 180,E1 -8160.643,E2 -8160.643} C_VEL
LIN {X 0,Y 459.753,Z 650.875,A -85,B 0,C 180,E1 -8163.488,E2 -8163.488} C_VEL
LIN {X 0,Y 459.137,Z 649.851,A -85,B 0,C 180,E1 -8164.208,E2 -8164.208} C_VEL
LIN {X 0,Y 456.323,Z 648.351,A -85,B 0,C 180,E1 -8165.382,E2 -8165.382} C_VEL
LIN {X 0,Y 453.917,Z 647.172,A -85,B 0,C 180,E1 -8166.329,E2 -8166.329} C_VEL
LIN {X 0,Y 452.883,Z 646.199,A -85,B 0,C 180,E1 -8167.059,E2 -8167.059} C_VEL
LIN {X 0,Y 452.8,Z 645.846,A -85,B 0,C 180,E1 -8167.306,E2 -8167.306} C_VEL
LIN {X 0,Y 452.949,Z 641.874,A -85,B 0,C 180,E1 -8170.04,E2 -8170.04} C_VEL
LIN {X 0,Y 453.082,Z 637.851,A -85,B 0,C 180,E1 -8172.859,E2 -8172.859} C_VEL
LIN {X 0,Y 453.217,Z 633.965,A -85,B 0,C 180,E1 -8175.634,E2 -8175.634} C_VEL
LIN {X 0,Y 453.388,Z 630.188,A -85,B 0,C 180,E1 -8178.374,E2 -8178.374} C_VEL
LIN {X 0,Y 453.391,Z 628.011,A -85,B 0,C 180,E1 -8180.182,E2 -8180.182} C_VEL
LIN {X 0,Y 453.639,Z 627.98,A -85,B 0,C 180,E1 -8182.88,E2 -8182.88} C_VEL
LIN {X 0,Y 453.673,Z 627.975,A -85,B 0,C 180,E1 -8184.666,E2 -8184.666} C_VEL
LIN {X 0,Y 453.768,Z 627.962,A -85,B 0,C 180,E1 -8187.336,E2 -8187.336} C_VEL
LIN {X 0,Y 453.828,Z 627.954,A -85,B 0,C 180,E1 -8190,E2 -8190} C_VEL
LIN {X 0,Y 453.768,Z 627.964,A -85,B 0,C 180,E1 -8192.663,E2 -8192.663} C_VEL
LIN {X 0,Y 453.667,Z 627.974,A -85,B 0,C 180,E1 -8196.225,E2 -8196.225} C_VEL
LIN {X 0,Y 453.563,Z 627.987,A -85,B 0,C 180,E1 -8198.016,E2 -8198.016} C_VEL
LIN {X 0,Y 453.199,Z 628.036,A -85,B 0,C 180,E1 -8201.177,E2 -8201.177} C_VEL
LIN {X 0,Y 453.063,Z 628.289,A -85,B 0,C 180,E1 -8201.633,E2 -8201.633} C_VEL
LIN {X 0,Y 452.934,Z 634.245,A -85,B 0,C 180,E1 -8205.294,E2 -8205.294} C_VEL
LIN {X 0,Y 452.807,Z 639.874,A -85,B 0,C 180,E1 -8208.776,E2 -8208.776} C_VEL
LIN {X 0,Y 452.693,Z 644.872,A -85,B 0,C 180,E1 -8211.875,E2 -8211.875} C_VEL
LIN {X 0,Y 452.611,Z 649.549,A -85,B 0,C 180,E1 -8214.787,E2 -8214.787} C_VEL
LIN {X 0,Y 452.572,Z 655.042,A -85,B 0,C 180,E1 -8218.207,E2 -8218.207} C_VEL
LIN {X 0,Y 455.461,Z 668.956,A -85,B 0,C 180,E1 -8218.734,E2 -8218.734} C_VEL
LIN {X 0,Y 456.368,Z 675.015,A -85,B 0,C 180,E1 -8219.018,E2 -8219.018} C_VEL
LIN {X 0,Y 455.833,Z 687.61,A -85,B 0,C 180,E1 -8219.669,E2 -8219.669} C_VEL
LIN {X 0,Y 455.281,Z 699.811,A -85,B 0,C 180,E1 -8220.505,E2 -8220.505} C_VEL
LIN {X 0,Y 454.747,Z 710.444,A -85,B 0,C 180,E1 -8221.439,E2 -8221.439} C_VEL
LIN {X 0,Y 454.199,Z 720.471,A -85,B 0,C 180,E1 -8222.526,E2 -8222.526} C_VEL
LIN {X 0,Y 453.67,Z 729.416,A -85,B 0,C 180,E1 -8223.721,E2 -8223.721} C_VEL
LIN {X 0,Y 453.272,Z 737.188,A -85,B 0,C 180,E1 -8225.007,E2 -8225.007} C_VEL
LIN {X 0,Y 452.943,Z 744.073,A -85,B 0,C 180,E1 -8226.422,E2 -8226.422} C_VEL
LIN {X 0,Y 452.697,Z 749.988,A -85,B 0,C 180,E1 -8227.991,E2 -8227.991} C_VEL
LIN {X 0,Y 452.497,Z 754.328,A -85,B 0,C 180,E1 -8229.552,E2 -8229.552} C_VEL
LIN {X 0,Y 452.374,Z 756.7,A -85,B 0,C 180,E1 -8230.73,E2 -8230.73} C_VEL
LIN {X 0,Y 452.345,Z 758.359,A -85,B 0,C 180,E1 -8231.918,E2 -8231.918} C_VEL
LIN {X 0,Y 452.326,Z 759.271,A -85,B 0,C 180,E1 -8233.129,E2 -8233.129} C_VEL
LIN {X 0,Y 452.347,Z 759.457,A -85,B 0,C 180,E1 -8234.382,E2 -8234.382} C_VEL
LIN {X 0,Y 452.349,Z 758.864,A -85,B 0,C 180,E1 -8235.641,E2 -8235.641} C_VEL
LIN {X 0,Y 452.391,Z 757.481,A -85,B 0,C 180,E1 -8236.899,E2 -8236.899} C_VEL
LIN {X 0,Y 452.493,Z 755.162,A -85,B 0,C 180,E1 -8238.203,E2 -8238.203} C_VEL
LIN {X 0,Y 452.653,Z 751.831,A -85,B 0,C 180,E1 -8239.533,E2 -8239.533} C_VEL
LIN {X 0,Y 452.828,Z 747.315,A -85,B 0,C 180,E1 -8240.896,E2 -8240.896} C_VEL
LIN {X 0,Y 453.079,Z 741.392,A -85,B 0,C 180,E1 -8242.287,E2 -8242.287} C_VEL
LIN {X 0,Y 453.483,Z 733.843,A -85,B 0,C 180,E1 -8243.695,E2 -8243.695} C_VEL
LIN {X 0,Y 453.906,Z 725.781,A -85,B 0,C 180,E1 -8244.913,E2 -8244.913} C_VEL
LIN {X 0,Y 454.455,Z 716.604,A -85,B 0,C 180,E1 -8246.036,E2 -8246.036} C_VEL
LIN {X 0,Y 454.984,Z 706.608,A -85,B 0,C 180,E1 -8247.033,E2 -8247.033} C_VEL
LIN {X 0,Y 455.544,Z 695.409,A -85,B 0,C 180,E1 -8247.933,E2 -8247.933} C_VEL
LIN {X 0,Y 456.071,Z 683.714,A -85,B 0,C 180,E1 -8248.662,E2 -8248.662} C_VEL
LIN {X 0,Y 456.31,Z 674.159,A -85,B 0,C 180,E1 -8249.131,E2 -8249.131} C_VEL
LIN {X 0,Y 454.16,Z 662.283,A -85,B 0,C 180,E1 -8249.645,E2 -8249.645} C_VEL
LIN {X 0,Y 452.594,Z 655.282,A -85,B 0,C 180,E1 -8249.916,E2 -8249.916} C_VEL
LIN {X 0,Y 452.675,Z 649.885,A -85,B 0,C 180,E1 -8253.241,E2 -8253.241} C_VEL
LIN {X 0,Y 452.725,Z 644.808,A -85,B 0,C 180,E1 -8256.333,E2 -8256.333} C_VEL
LIN {X 0,Y 452.811,Z 640.353,A -85,B 0,C 180,E1 -8259.085,E2 -8259.085} C_VEL
LIN {X 0,Y 452.878,Z 635.524,A -85,B 0,C 180,E1 -8261.918,E2 -8261.918} C_VEL
LIN {X 0,Y 452.957,Z 630.698,A -85,B 0,C 180,E1 -8264.706,E2 -8264.706} C_VEL
LIN {X 0,Y 452.995,Z 628.064,A -85,B 0,C 180,E1 -8266.314,E2 -8266.314} C_VEL
LIN {X 0,Y 453.382,Z 628.014,A -85,B 0,C 180,E1 -8268.374,E2 -8268.374} C_VEL
LIN {X 0,Y 453.583,Z 627.989,A -85,B 0,C 180,E1 -8271.086,E2 -8271.086} C_VEL
LIN {X 0,Y 453.674,Z 627.977,A -85,B 0,C 180,E1 -8273.775,E2 -8273.775} C_VEL
LIN {X 0,Y 453.763,Z 627.965,A -85,B 0,C 180,E1 -8277.337,E2 -8277.337} C_VEL
LIN {X 0,Y 453.82,Z 627.958,A -85,B 0,C 180,E1 -8280,E2 -8280} C_VEL
LIN {X 0,Y 453.762,Z 627.965,A -85,B 0,C 180,E1 -8282.663,E2 -8282.663} C_VEL
LIN {X 0,Y 453.674,Z 627.975,A -85,B 0,C 180,E1 -8286.225,E2 -8286.225} C_VEL
LIN {X 0,Y 453.59,Z 627.986,A -85,B 0,C 180,E1 -8288.913,E2 -8288.913} C_VEL
LIN {X 0,Y 453.559,Z 627.99,A -85,B 0,C 180,E1 -8292.529,E2 -8292.529} C_VEL
LIN {X 0,Y 453.541,Z 627.991,A -85,B 0,C 180,E1 -8296.196,E2 -8296.196} C_VEL
LIN {X 0,Y 453.517,Z 627.994,A -85,B 0,C 180,E1 -8299.041,E2 -8299.041} C_VEL
LIN {X 0,Y 453.473,Z 628,A -85,B 0,C 180,E1 -8301.836,E2 -8301.836} C_VEL
LIN {X 0,Y 453.511,Z 627.995,A -85,B 0,C 180,E1 -8304.735,E2 -8304.735} C_VEL
LIN {X 0,Y 453.536,Z 627.994,A -85,B 0,C 180,E1 -8307.962,E2 -8307.962} C_VEL
LIN {X 0,Y 453.48,Z 627.998,A -85,B 0,C 180,E1 -8310.759,E2 -8310.759} C_VEL
LIN {X 0,Y 453.475,Z 628,A -85,B 0,C 180,E1 -8313.913,E2 -8313.913} C_VEL
LIN {X 0,Y 453.467,Z 628.002,A -85,B 0,C 180,E1 -8317.188,E2 -8317.188} C_VEL
LIN {X 0,Y 453.503,Z 627.997,A -85,B 0,C 180,E1 -8319.449,E2 -8319.449} C_VEL
LIN {X 0,Y 453.461,Z 628.002,A -85,B 0,C 180,E1 -8322.995,E2 -8322.995} C_VEL
LIN {X 0,Y 453.464,Z 628.002,A -85,B 0,C 180,E1 -8325.78,E2 -8325.78} C_VEL
LIN {X 0,Y 453.477,Z 628,A -85,B 0,C 180,E1 -8328.21,E2 -8328.21} C_VEL
LIN {X 0,Y 453.547,Z 628.134,A -85,B 0,C 180,E1 -8330.485,E2 -8330.485} C_VEL
LIN {X 0,Y 454.424,Z 633.912,A -85,B 0,C 180,E1 -8333.535,E2 -8333.535} C_VEL
LIN {X 0,Y 454.488,Z 638.148,A -85,B 0,C 180,E1 -8335.639,E2 -8335.639} C_VEL
LIN {X 0,Y 454.112,Z 644.809,A -85,B 0,C 180,E1 -8338.808,E2 -8338.808} C_VEL
LIN {X 0,Y 453.784,Z 651.706,A -85,B 0,C 180,E1 -8341.981,E2 -8341.981} C_VEL
LIN {X 0,Y 453.468,Z 659.073,A -85,B 0,C 180,E1 -8345.264,E2 -8345.264} C_VEL
LIN {X 0,Y 453.222,Z 666.499,A -85,B 0,C 180,E1 -8348.499,E2 -8348.499} C_VEL
LIN {X 0,Y 453.004,Z 672.724,A -85,B 0,C 180,E1 -8351.15,E2 -8351.15} C_VEL
LIN {X 0,Y 452.874,Z 679.811,A -85,B 0,C 180,E1 -8354.119,E2 -8354.119} C_VEL
LIN {X 0,Y 455.213,Z 694.166,A -85,B 0,C 180,E1 -8354.618,E2 -8354.618} C_VEL
LIN {X 0,Y 456.188,Z 702.406,A -85,B 0,C 180,E1 -8354.989,E2 -8354.989} C_VEL
LIN {X 0,Y 455.689,Z 714.183,A -85,B 0,C 180,E1 -8355.6,E2 -8355.6} C_VEL
LIN {X 0,Y 455.147,Z 725.619,A -85,B 0,C 180,E1 -8356.381,E2 -8356.381} C_VEL
LIN {X 0,Y 454.659,Z 736.773,A -85,B 0,C 180,E1 -8357.345,E2 -8357.345} C_VEL
LIN {X 0,Y 454.056,Z 746.599,A -85,B 0,C 180,E1 -8358.392,E2 -8358.392} C_VEL
LIN {X 0,Y 453.564,Z 755.148,A -85,B 0,C 180,E1 -8359.51,E2 -8359.51} C_VEL
LIN {X 0,Y 453.152,Z 763.472,A -85,B 0,C 180,E1 -8360.853,E2 -8360.853} C_VEL
LIN {X 0,Y 452.844,Z 770.182,A -85,B 0,C 180,E1 -8362.196,E2 -8362.196} C_VEL
LIN {X 0,Y 452.632,Z 776.329,A -85,B 0,C 180,E1 -8363.761,E2 -8363.761} C_VEL
LIN {X 0,Y 452.562,Z 780.317,A -85,B 0,C 180,E1 -8365.101,E2 -8365.101} C_VEL
LIN {X 0,Y 452.486,Z 783.259,A -85,B 0,C 180,E1 -8366.438,E2 -8366.438} C_VEL
LIN {X 0,Y 452.495,Z 784.661,A -85,B 0,C 180,E1 -8367.33,E2 -8367.33} C_VEL
LIN {X 0,Y 452.428,Z 786.262,A -85,B 0,C 180,E1 -8369.11,E2 -8369.11} C_VEL
LIN {X 0,Y 452.434,Z 786.474,A -85,B 0,C 180,E1 -8370,E2 -8370} C_VEL
LIN {X 0,Y 452.428,Z 786.251,A -85,B 0,C 180,E1 -8370.89,E2 -8370.89} C_VEL
LIN {X 0,Y 452.495,Z 784.627,A -85,B 0,C 180,E1 -8372.671,E2 -8372.671} C_VEL
LIN {X 0,Y 452.486,Z 783.214,A -85,B 0,C 180,E1 -8373.562,E2 -8373.562} C_VEL
LIN {X 0,Y 452.562,Z 780.25,A -85,B 0,C 180,E1 -8374.9,E2 -8374.9} C_VEL
LIN {X 0,Y 452.691,Z 775.364,A -85,B 0,C 180,E1 -8376.486,E2 -8376.486} C_VEL
LIN {X 0,Y 452.898,Z 769.056,A -85,B 0,C 180,E1 -8378.029,E2 -8378.029} C_VEL
LIN {X 0,Y 453.223,Z 762.1,A -85,B 0,C 180,E1 -8379.371,E2 -8379.371} C_VEL
LIN {X 0,Y 453.637,Z 753.391,A -85,B 0,C 180,E1 -8380.715,E2 -8380.715} C_VEL
LIN {X 0,Y 454.181,Z 744.477,A -85,B 0,C 180,E1 -8381.832,E2 -8381.832} C_VEL
LIN {X 0,Y 454.683,Z 733.963,A -85,B 0,C 180,E1 -8382.909,E2 -8382.909} C_VEL
LIN {X 0,Y 455.219,Z 722.432,A -85,B 0,C 180,E1 -8383.846,E2 -8383.846} C_VEL
LIN {X 0,Y 455.836,Z 710.072,A -85,B 0,C 180,E1 -8384.624,E2 -8384.624} C_VEL
LIN {X 0,Y 456.165,Z 700.968,A -85,B 0,C 180,E1 -8385.07,E2 -8385.07} C_VEL
LIN {X 0,Y 454.202,Z 687.429,A -85,B 0,C 180,E1 -8385.639,E2 -8385.639} C_VEL
LIN {X 0,Y 452.858,Z 679.419,A -85,B 0,C 180,E1 -8385.9,E2 -8385.9} C_VEL
LIN {X 0,Y 453.072,Z 670.838,A -85,B 0,C 180,E1 -8389.482,E2 -8389.482} C_VEL
LIN {X 0,Y 453.259,Z 664.18,A -85,B 0,C 180,E1 -8392.327,E2 -8392.327} C_VEL
LIN {X 0,Y 453.527,Z 656.441,A -85,B 0,C 180,E1 -8395.715,E2 -8395.715} C_VEL
LIN {X 0,Y 453.822,Z 649.886,A -85,B 0,C 180,E1 -8398.69,E2 -8398.69} C_VEL
LIN {X 0,Y 454.14,Z 643.443,A -85,B 0,C 180,E1 -8401.747,E2 -8401.747} C_VEL
LIN {X 0,Y 454.541,Z 637.093,A -85,B 0,C 180,E1 -8404.896,E2 -8404.896} C_VEL
LIN {X 0,Y 454.316,Z 632.943,A -85,B 0,C 180,E1 -8407.107,E2 -8407.107} C_VEL
LIN {X 0,Y 453.511,Z 627.998,A -85,B 0,C 180,E1 -8410.025,E2 -8410.025} C_VEL
LIN {X 0,Y 453.466,Z 628.003,A -85,B 0,C 180,E1 -8413.245,E2 -8413.245} C_VEL
LIN {X 0,Y 453.468,Z 628.001,A -85,B 0,C 180,E1 -8415.779,E2 -8415.779} C_VEL
LIN {X 0,Y 453.481,Z 628.001,A -85,B 0,C 180,E1 -8418.209,E2 -8418.209} C_VEL
LIN {X 0,Y 453.496,Z 627.999,A -85,B 0,C 180,E1 -8420.793,E2 -8420.793} C_VEL
LIN {X 0,Y 453.457,Z 628.003,A -85,B 0,C 180,E1 -8423.917,E2 -8423.917} C_VEL
LIN {X 0,Y 453.485,Z 628,A -85,B 0,C 180,E1 -8427.151,E2 -8427.151} C_VEL
LIN {X 0,Y 453.477,Z 628,A -85,B 0,C 180,E1 -8430.268,E2 -8430.268} C_VEL
LIN {X 0,Y 453.508,Z 627.997,A -85,B 0,C 180,E1 -8433.294,E2 -8433.294} C_VEL
LIN {X 0,Y 453.505,Z 627.994,A -85,B 0,C 180,E1 -8436.239,E2 -8436.239} C_VEL
LIN {X 0,Y 453.484,Z 627.998,A -85,B 0,C 180,E1 -8439.118,E2 -8439.118} C_VEL
LIN {X 0,Y 453.513,Z 627.996,A -85,B 0,C 180,E1 -8441.945,E2 -8441.945} C_VEL
LIN {X 0,Y 453.541,Z 627.992,A -85,B 0,C 180,E1 -8444.726,E2 -8444.726} C_VEL
LIN {X 0,Y 453.561,Z 627.99,A -85,B 0,C 180,E1 -8448.379,E2 -8448.379} C_VEL
LIN {X 0,Y 453.654,Z 627.976,A -85,B 0,C 180,E1 -8451.985,E2 -8451.985} C_VEL
LIN {X 0,Y 453.672,Z 627.976,A -85,B 0,C 180,E1 -8454.667,E2 -8454.667} C_VEL
LIN {X 0,Y 453.746,Z 627.966,A -85,B 0,C 180,E1 -8457.337,E2 -8457.337} C_VEL
LIN {X 0,Y 453.825,Z 627.957,A -85,B 0,C 180,E1 -8460,E2 -8460} C_VEL
LIN {X 0,Y 453.767,Z 627.966,A -85,B 0,C 180,E1 -8462.663,E2 -8462.663} C_VEL
LIN {X 0,Y 453.679,Z 627.975,A -85,B 0,C 180,E1 -8466.225,E2 -8466.225} C_VEL
LIN {X 0,Y 453.647,Z 627.981,A -85,B 0,C 180,E1 -8468.015,E2 -8468.015} C_VEL
LIN {X 0,Y 453.538,Z 627.994,A -85,B 0,C 180,E1 -8468.915,E2 -8468.915} C_VEL
LIN {X 0,Y 453.508,Z 630.018,A -85,B 0,C 180,E1 -8470.717,E2 -8470.717} C_VEL
LIN {X 0,Y 453.323,Z 633.588,A -85,B 0,C 180,E1 -8473.447,E2 -8473.447} C_VEL
LIN {X 0,Y 453.189,Z 637.276,A -85,B 0,C 180,E1 -8476.209,E2 -8476.209} C_VEL
LIN {X 0,Y 453.104,Z 641.14,A -85,B 0,C 180,E1 -8479.01,E2 -8479.01} C_VEL
LIN {X 0,Y 452.916,Z 645.156,A -85,B 0,C 180,E1 -8481.865,E2 -8481.865} C_VEL
LIN {X 0,Y 452.824,Z 649.314,A -85,B 0,C 180,E1 -8484.775,E2 -8484.775} C_VEL
LIN {X 0,Y 452.694,Z 653.67,A -85,B 0,C 180,E1 -8487.759,E2 -8487.759} C_VEL
LIN {X 0,Y 452.624,Z 655.796,A -85,B 0,C 180,E1 -8489.187,E2 -8489.187} C_VEL
LIN {X 0,Y 455.574,Z 669.174,A -85,B 0,C 180,E1 -8489.709,E2 -8489.709} C_VEL
LIN {X 0,Y 456.414,Z 674.868,A -85,B 0,C 180,E1 -8489.974,E2 -8489.974} C_VEL
LIN {X 0,Y 455.909,Z 687.9,A -85,B 0,C 180,E1 -8490.642,E2 -8490.642} C_VEL
LIN {X 0,Y 455.399,Z 698.874,A -85,B 0,C 180,E1 -8491.39,E2 -8491.39} C_VEL
LIN {X 0,Y 454.784,Z 710.48,A -85,B 0,C 180,E1 -8492.393,E2 -8492.393} C_VEL
LIN {X 0,Y 454.29,Z 719.362,A -85,B 0,C 180,E1 -8493.343,E2 -8493.343} C_VEL
LIN {X 0,Y 453.887,Z 727.65,A -85,B 0,C 180,E1 -8494.414,E2 -8494.414} C_VEL
LIN {X 0,Y 453.463,Z 734.853,A -85,B 0,C 180,E1 -8495.535,E2 -8495.535} C_VEL
LIN {X 0,Y 453.064,Z 742.336,A -85,B 0,C 180,E1 -8496.971,E2 -8496.971} C_VEL
LIN {X 0,Y 452.788,Z 748.108,A -85,B 0,C 180,E1 -8498.379,E2 -8498.379} C_VEL
LIN {X 0,Y 452.629,Z 753.147,A -85,B 0,C 180,E1 -8499.993,E2 -8499.993} C_VEL
LIN {X 0,Y 452.523,Z 755.992,A -85,B 0,C 180,E1 -8501.248,E2 -8501.248} C_VEL
LIN {X 0,Y 452.451,Z 757.148,A -85,B 0,C 180,E1 -8501.907,E2 -8501.907} C_VEL
LIN {X 0,Y 452.366,Z 758.691,A -85,B 0,C 180,E1 -8503.125,E2 -8503.125} C_VEL
LIN {X 0,Y 452.353,Z 759.509,A -85,B 0,C 180,E1 -8504.383,E2 -8504.383} C_VEL
LIN {X 0,Y 452.351,Z 759.51,A -85,B 0,C 180,E1 -8505.641,E2 -8505.641} C_VEL
LIN {X 0,Y 452.346,Z 758.711,A -85,B 0,C 180,E1 -8506.906,E2 -8506.906} C_VEL
LIN {X 0,Y 452.441,Z 757.045,A -85,B 0,C 180,E1 -8508.212,E2 -8508.212} C_VEL
LIN {X 0,Y 452.573,Z 754.42,A -85,B 0,C 180,E1 -8509.546,E2 -8509.546} C_VEL
LIN {X 0,Y 452.684,Z 750.672,A -85,B 0,C 180,E1 -8510.92,E2 -8510.92} C_VEL
LIN {X 0,Y 452.894,Z 745.652,A -85,B 0,C 180,E1 -8512.318,E2 -8512.318} C_VEL
LIN {X 0,Y 453.176,Z 739.112,A -85,B 0,C 180,E1 -8513.749,E2 -8513.749} C_VEL
LIN {X 0,Y 453.598,Z 731.849,A -85,B 0,C 180,E1 -8515.021,E2 -8515.021} C_VEL
LIN {X 0,Y 454.106,Z 722.882,A -85,B 0,C 180,E1 -8516.286,E2 -8516.286} C_VEL
LIN {X 0,Y 454.599,Z 713.548,A -85,B 0,C 180,E1 -8517.36,E2 -8517.36} C_VEL
LIN {X 0,Y 455.18,Z 703.135,A -85,B 0,C 180,E1 -8518.334,E2 -8518.334} C_VEL
LIN {X 0,Y 455.657,Z 692.306,A -85,B 0,C 180,E1 -8519.146,E2 -8519.146} C_VEL
LIN {X 0,Y 456.224,Z 679.369,A -85,B 0,C 180,E1 -8519.887,E2 -8519.887} C_VEL
LIN {X 0,Y 456.257,Z 673.367,A -85,B 0,C 180,E1 -8520.167,E2 -8520.167} C_VEL
LIN {X 0,Y 453.78,Z 660.795,A -85,B 0,C 180,E1 -8520.707,E2 -8520.707} C_VEL
LIN {X 0,Y 452.594,Z 655.35,A -85,B 0,C 180,E1 -8520.907,E2 -8520.907} C_VEL
LIN {X 0,Y 452.718,Z 650.412,A -85,B 0,C 180,E1 -8524.21,E2 -8524.21} C_VEL
LIN {X 0,Y 452.8,Z 645.846,A -85,B 0,C 180,E1 -8527.306,E2 -8527.306} C_VEL
LIN {X 0,Y 452.147,Z 644.844,A -85,B 0,C 180,E1 -8528.038,E2 -8528.038} C_VEL
LIN {X 0,Y 449.344,Z 643.396,A -85,B 0,C 180,E1 -8529.233,E2 -8529.233} C_VEL
LIN {X 0,Y 446.989,Z 642.263,A -85,B 0,C 180,E1 -8530.198,E2 -8530.198} C_VEL
LIN {X 0,Y 445.999,Z 641.313,A -85,B 0,C 180,E1 -8530.941,E2 -8530.941} C_VEL
LIN {X 0,Y 445.93,Z 640.964,A -85,B 0,C 180,E1 -8531.191,E2 -8531.191} C_VEL
LIN {X 0,Y 446.115,Z 636.385,A -85,B 0,C 180,E1 -8534.465,E2 -8534.465} C_VEL
LIN {X 0,Y 446.287,Z 632.201,A -85,B 0,C 180,E1 -8537.518,E2 -8537.518} C_VEL
LIN {X 0,Y 446.328,Z 628.891,A -85,B 0,C 180,E1 -8540.025,E2 -8540.025} C_VEL
LIN {X 0,Y 446.608,Z 628.857,A -85,B 0,C 180,E1 -8542.767,E2 -8542.767} C_VEL
LIN {X 0,Y 446.648,Z 628.85,A -85,B 0,C 180,E1 -8544.582,E2 -8544.582} C_VEL
LIN {X 0,Y 446.712,Z 628.842,A -85,B 0,C 180,E1 -8547.294,E2 -8547.294} C_VEL
LIN {X 0,Y 446.798,Z 628.829,A -85,B 0,C 180,E1 -8550,E2 -8550} C_VEL
LIN {X 0,Y 446.712,Z 628.843,A -85,B 0,C 180,E1 -8552.705,E2 -8552.705} C_VEL
LIN {X 0,Y 446.636,Z 628.85,A -85,B 0,C 180,E1 -8556.323,E2 -8556.323} C_VEL
LIN {X 0,Y 446.422,Z 628.88,A -85,B 0,C 180,E1 -8559.057,E2 -8559.057} C_VEL
LIN {X 0,Y 446.004,Z 628.956,A -85,B 0,C 180,E1 -8561.59,E2 -8561.59} C_VEL
LIN {X 0,Y 445.854,Z 633.827,A -85,B 0,C 180,E1 -8564.608,E2 -8564.608} C_VEL
LIN {X 0,Y 445.754,Z 638.38,A -85,B 0,C 180,E1 -8567.431,E2 -8567.431} C_VEL
LIN {X 0,Y 445.655,Z 642.966,A -85,B 0,C 180,E1 -8570.3,E2 -8570.3} C_VEL
LIN {X 0,Y 445.585,Z 648.595,A -85,B 0,C 180,E1 -8573.821,E2 -8573.821} C_VEL
LIN {X 0,Y 445.512,Z 652.412,A -85,B 0,C 180,E1 -8576.212,E2 -8576.212} C_VEL
LIN {X 0,Y 445.529,Z 655.352,A -85,B 0,C 180,E1 -8577.968,E2 -8577.968} C_VEL
LIN {X 0,Y 448.341,Z 668.598,A -85,B 0,C 180,E1 -8578.472,E2 -8578.472} C_VEL
LIN {X 0,Y 449.497,Z 675.699,A -85,B 0,C 180,E1 -8578.814,E2 -8578.814} C_VEL
LIN {X 0,Y 448.926,Z 688.303,A -85,B 0,C 180,E1 -8579.482,E2 -8579.482} C_VEL
LIN {X 0,Y 448.34,Z 700.561,A -85,B 0,C 180,E1 -8580.346,E2 -8580.346} C_VEL
LIN {X 0,Y 447.758,Z 711.37,A -85,B 0,C 180,E1 -8581.322,E2 -8581.322} C_VEL
LIN {X 0,Y 447.203,Z 721.314,A -85,B 0,C 180,E1 -8582.431,E2 -8582.431} C_VEL
LIN {X 0,Y 446.628,Z 730.473,A -85,B 0,C 180,E1 -8583.701,E2 -8583.701} C_VEL
LIN {X 0,Y 446.209,Z 738.131,A -85,B 0,C 180,E1 -8585.012,E2 -8585.012} C_VEL
LIN {X 0,Y 445.875,Z 745.075,A -85,B 0,C 180,E1 -8586.498,E2 -8586.498} C_VEL
LIN {X 0,Y 445.615,Z 750.357,A -85,B 0,C 180,E1 -8587.958,E2 -8587.958} C_VEL
LIN {X 0,Y 445.426,Z 754.238,A -85,B 0,C 180,E1 -8589.364,E2 -8589.364} C_VEL
LIN {X 0,Y 445.288,Z 756.998,A -85,B 0,C 180,E1 -8590.748,E2 -8590.748} C_VEL
LIN {X 0,Y 445.248,Z 758.756,A -85,B 0,C 180,E1 -8592.109,E2 -8592.109} C_VEL
LIN {X 0,Y 445.253,Z 759.7,A -85,B 0,C 180,E1 -8593.987,E2 -8593.987} C_VEL
LIN {X 0,Y 445.274,Z 759.339,A -85,B 0,C 180,E1 -8595.255,E2 -8595.255} C_VEL
LIN {X 0,Y 445.267,Z 758.17,A -85,B 0,C 180,E1 -8596.556,E2 -8596.556} C_VEL
LIN {X 0,Y 445.377,Z 756.132,A -85,B 0,C 180,E1 -8597.872,E2 -8597.872} C_VEL
LIN {X 0,Y 445.542,Z 753.121,A -85,B 0,C 180,E1 -8599.213,E2 -8599.213} C_VEL
LIN {X 0,Y 445.748,Z 747.89,A -85,B 0,C 180,E1 -8600.9,E2 -8600.9} C_VEL
LIN {X 0,Y 446.033,Z 741.822,A -85,B 0,C 180,E1 -8602.369,E2 -8602.369} C_VEL
LIN {X 0,Y 446.394,Z 735.083,A -85,B 0,C 180,E1 -8603.668,E2 -8603.668} C_VEL
LIN {X 0,Y 446.91,Z 726.263,A -85,B 0,C 180,E1 -8605.043,E2 -8605.043} C_VEL
LIN {X 0,Y 447.508,Z 716.848,A -85,B 0,C 180,E1 -8606.219,E2 -8606.219} C_VEL
LIN {X 0,Y 448.093,Z 706.755,A -85,B 0,C 180,E1 -8607.241,E2 -8607.241} C_VEL
LIN {X 0,Y 448.598,Z 696.573,A -85,B 0,C 180,E1 -8608.079,E2 -8608.079} C_VEL
LIN {X 0,Y 449.169,Z 684.751,A -85,B 0,C 180,E1 -8608.847,E2 -8608.847} C_VEL
LIN {X 0,Y 449.519,Z 675.713,A -85,B 0,C 180,E1 -8609.304,E2 -8609.304} C_VEL
LIN {X 0,Y 447.512,Z 664.335,A -85,B 0,C 180,E1 -8609.831,E2 -8609.831} C_VEL
LIN {X 0,Y 445.537,Z 655.575,A -85,B 0,C 180,E1 -8610.15,E2 -8610.15} C_VEL
LIN {X 0,Y 445.575,Z 651.266,A -85,B 0,C 180,E1 -8612.78,E2 -8612.78} C_VEL
LIN {X 0,Y 445.626,Z 646.379,A -85,B 0,C 180,E1 -8615.792,E2 -8615.792} C_VEL
LIN {X 0,Y 445.718,Z 641.578,A -85,B 0,C 180,E1 -8618.736,E2 -8618.736} C_VEL
LIN {X 0,Y 445.816,Z 636.807,A -85,B 0,C 180,E1 -8621.622,E2 -8621.622} C_VEL
LIN {X 0,Y 445.882,Z 631.892,A -85,B 0,C 180,E1 -8624.457,E2 -8624.457} C_VEL
LIN {X 0,Y 445.958,Z 628.941,A -85,B 0,C 180,E1 -8626.21,E2 -8626.21} C_VEL
LIN {X 0,Y 446.326,Z 628.892,A -85,B 0,C 180,E1 -8628.188,E2 -8628.188} C_VEL
LIN {X 0,Y 446.526,Z 628.868,A -85,B 0,C 180,E1 -8630.944,E2 -8630.944} C_VEL
LIN {X 0,Y 446.643,Z 628.852,A -85,B 0,C 180,E1 -8633.676,E2 -8633.676} C_VEL
LIN {X 0,Y 446.707,Z 628.844,A -85,B 0,C 180,E1 -8637.295,E2 -8637.295} C_VEL
LIN {X 0,Y 446.791,Z 628.833,A -85,B 0,C 180,E1 -8640,E2 -8640} C_VEL
LIN {X 0,Y 446.706,Z 628.844,A -85,B 0,C 180,E1 -8642.705,E2 -8642.705} C_VEL
LIN {X 0,Y 446.643,Z 628.852,A -85,B 0,C 180,E1 -8646.324,E2 -8646.324} C_VEL
LIN {X 0,Y 446.535,Z 628.864,A -85,B 0,C 180,E1 -8649.055,E2 -8649.055} C_VEL
LIN {X 0,Y 446.517,Z 628.868,A -85,B 0,C 180,E1 -8652.73,E2 -8652.73} C_VEL
LIN {X 0,Y 446.492,Z 628.869,A -85,B 0,C 180,E1 -8656.228,E2 -8656.228} C_VEL
LIN {X 0,Y 446.466,Z 628.872,A -85,B 0,C 180,E1 -8659.303,E2 -8659.303} C_VEL
LIN {X 0,Y 446.415,Z 628.88,A -85,B 0,C 180,E1 -8662.2,E2 -8662.2} C_VEL
LIN {X 0,Y 446.455,Z 628.875,A -85,B 0,C 180,E1 -8665.153,E2 -8665.153} C_VEL
LIN {X 0,Y 446.481,Z 628.871,A -85,B 0,C 180,E1 -8668.179,E2 -8668.179} C_VEL
LIN {X 0,Y 446.417,Z 628.88,A -85,B 0,C 180,E1 -8671.3,E2 -8671.3} C_VEL
LIN {X 0,Y 446.427,Z 628.878,A -85,B 0,C 180,E1 -8674.523,E2 -8674.523} C_VEL
LIN {X 0,Y 446.428,Z 628.877,A -85,B 0,C 180,E1 -8678.082,E2 -8678.082} C_VEL
LIN {X 0,Y 446.424,Z 628.878,A -85,B 0,C 180,E1 -8680.918,E2 -8680.918} C_VEL
LIN {X 0,Y 446.399,Z 628.882,A -85,B 0,C 180,E1 -8683.846,E2 -8683.846} C_VEL
LIN {X 0,Y 446.398,Z 628.882,A -85,B 0,C 180,E1 -8686.404,E2 -8686.404} C_VEL
LIN {X 0,Y 446.464,Z 628.874,A -85,B 0,C 180,E1 -8689.805,E2 -8689.805} C_VEL
LIN {X 0,Y 446.491,Z 629.003,A -85,B 0,C 180,E1 -8690.267,E2 -8690.267} C_VEL
LIN {X 0,Y 447.378,Z 634.729,A -85,B 0,C 180,E1 -8693.349,E2 -8693.349} C_VEL
LIN {X 0,Y 447.491,Z 639.122,A -85,B 0,C 180,E1 -8695.571,E2 -8695.571} C_VEL
LIN {X 0,Y 447.093,Z 645.706,A -85,B 0,C 180,E1 -8698.753,E2 -8698.753} C_VEL
LIN {X 0,Y 446.754,Z 652.295,A -85,B 0,C 180,E1 -8701.84,E2 -8701.84} C_VEL
LIN {X 0,Y 446.456,Z 658.905,A -85,B 0,C 180,E1 -8704.848,E2 -8704.848} C_VEL
LIN {X 0,Y 446.181,Z 666.768,A -85,B 0,C 180,E1 -8708.332,E2 -8708.332} C_VEL
LIN {X 0,Y 445.903,Z 674.365,A -85,B 0,C 180,E1 -8711.626,E2 -8711.626} C_VEL
LIN {X 0,Y 445.839,Z 679.826,A -85,B 0,C 180,E1 -8713.88,E2 -8713.88} C_VEL
LIN {X 0,Y 448.04,Z 693.116,A -85,B 0,C 180,E1 -8714.339,E2 -8714.339} C_VEL
LIN {X 0,Y 449.318,Z 702.082,A -85,B 0,C 180,E1 -8714.754,E2 -8714.754} C_VEL
LIN {X 0,Y 448.807,Z 713.887,A -85,B 0,C 180,E1 -8715.375,E2 -8715.375} C_VEL
LIN {X 0,Y 448.24,Z 725.341,A -85,B 0,C 180,E1 -8716.167,E2 -8716.167} C_VEL
LIN {X 0,Y 447.694,Z 735.301,A -85,B 0,C 180,E1 -8717.027,E2 -8717.027} C_VEL
LIN {X 0,Y 447.215,Z 744.387,A -85,B 0,C 180,E1 -8717.982,E2 -8717.982} C_VEL
LIN {X 0,Y 446.628,Z 753.292,A -85,B 0,C 180,E1 -8719.116,E2 -8719.116} C_VEL
LIN {X 0,Y 446.174,Z 761.994,A -85,B 0,C 180,E1 -8720.48,E2 -8720.48} C_VEL
LIN {X 0,Y 445.854,Z 768.937,A -85,B 0,C 180,E1 -8721.845,E2 -8721.845} C_VEL
LIN {X 0,Y 445.582,Z 774.5,A -85,B 0,C 180,E1 -8723.207,E2 -8723.207} C_VEL
LIN {X 0,Y 445.512,Z 778.865,A -85,B 0,C 180,E1 -8724.569,E2 -8724.569} C_VEL
LIN {X 0,Y 445.424,Z 781.17,A -85,B 0,C 180,E1 -8725.476,E2 -8725.476} C_VEL
LIN {X 0,Y 445.384,Z 783.042,A -85,B 0,C 180,E1 -8726.382,E2 -8726.382} C_VEL
LIN {X 0,Y 445.422,Z 784.448,A -85,B 0,C 180,E1 -8727.287,E2 -8727.287} C_VEL
LIN {X 0,Y 445.338,Z 786.05,A -85,B 0,C 180,E1 -8729.096,E2 -8729.096} C_VEL
LIN {X 0,Y 445.342,Z 786.264,A -85,B 0,C 180,E1 -8730,E2 -8730} C_VEL
LIN {X 0,Y 445.338,Z 786.041,A -85,B 0,C 180,E1 -8730.905,E2 -8730.905} C_VEL
LIN {X 0,Y 445.422,Z 784.416,A -85,B 0,C 180,E1 -8732.713,E2 -8732.713} C_VEL
LIN {X 0,Y 445.385,Z 783.001,A -85,B 0,C 180,E1 -8733.619,E2 -8733.619} C_VEL
LIN {X 0,Y 445.493,Z 780.036,A -85,B 0,C 180,E1 -8734.978,E2 -8734.978} C_VEL
LIN {X 0,Y 445.584,Z 775.655,A -85,B 0,C 180,E1 -8736.448,E2 -8736.448} C_VEL
LIN {X 0,Y 445.774,Z 769.852,A -85,B 0,C 180,E1 -8737.93,E2 -8737.93} C_VEL
LIN {X 0,Y 446.107,Z 763.117,A -85,B 0,C 180,E1 -8739.293,E2 -8739.293} C_VEL
LIN {X 0,Y 446.536,Z 754.767,A -85,B 0,C 180,E1 -8740.658,E2 -8740.658} C_VEL
LIN {X 0,Y 447.073,Z 746.202,A -85,B 0,C 180,E1 -8741.792,E2 -8741.792} C_VEL
LIN {X 0,Y 447.651,Z 736.642,A -85,B 0,C 180,E1 -8742.83,E2 -8742.83} C_VEL
LIN {X 0,Y 448.095,Z 726.624,A -85,B 0,C 180,E1 -8743.723,E2 -8743.723} C_VEL
LIN {X 0,Y 448.673,Z 715.556,A -85,B 0,C 180,E1 -8744.515,E2 -8744.515} C_VEL
LIN {X 0,Y 449.259,Z 703.328,A -85,B 0,C 180,E1 -8745.191,E2 -8745.191} C_VEL
LIN {X 0,Y 447.895,Z 692.161,A -85,B 0,C 180,E1 -8745.709,E2 -8745.709} C_VEL
LIN {X 0,Y 445.781,Z 679.196,A -85,B 0,C 180,E1 -8746.166,E2 -8746.166} C_VEL
LIN {X 0,Y 446.029,Z 670.659,A -85,B 0,C 180,E1 -8749.802,E2 -8749.802} C_VEL
LIN {X 0,Y 446.192,Z 664.023,A -85,B 0,C 180,E1 -8752.7,E2 -8752.7} C_VEL
LIN {X 0,Y 446.462,Z 657.43,A -85,B 0,C 180,E1 -8755.651,E2 -8755.651} C_VEL
LIN {X 0,Y 446.73,Z 651.804,A -85,B 0,C 180,E1 -8758.237,E2 -8758.237} C_VEL
LIN {X 0,Y 447.051,Z 645.512,A -85,B 0,C 180,E1 -8761.251,E2 -8761.251} C_VEL
LIN {X 0,Y 447.479,Z 639.171,A -85,B 0,C 180,E1 -8764.431,E2 -8764.431} C_VEL
LIN {X 0,Y 447.387,Z 634.815,A -85,B 0,C 180,E1 -8766.759,E2 -8766.759} C_VEL
LIN {X 0,Y 446.677,Z 629.998,A -85,B 0,C 180,E1 -8769.559,E2 -8769.559} C_VEL
LIN {X 0,Y 446.476,Z 628.875,A -85,B 0,C 180,E1 -8770.331,E2 -8770.331} C_VEL
LIN {X 0,Y 446.425,Z 628.879,A -85,B 0,C 180,E1 -8773.843,E2 -8773.843} C_VEL
LIN {X 0,Y 446.401,Z 628.883,A -85,B 0,C 180,E1 -8776.403,E2 -8776.403} C_VEL
LIN {X 0,Y 446.429,Z 628.88,A -85,B 0,C 180,E1 -8779.082,E2 -8779.082} C_VEL
LIN {X 0,Y 446.417,Z 628.88,A -85,B 0,C 180,E1 -8781.921,E2 -8781.921} C_VEL
LIN {X 0,Y 446.431,Z 628.878,A -85,B 0,C 180,E1 -8785.477,E2 -8785.477} C_VEL
LIN {X 0,Y 446.418,Z 628.88,A -85,B 0,C 180,E1 -8788.7,E2 -8788.7} C_VEL
LIN {X 0,Y 446.486,Z 628.87,A -85,B 0,C 180,E1 -8791.821,E2 -8791.821} C_VEL
LIN {X 0,Y 446.459,Z 628.874,A -85,B 0,C 180,E1 -8794.848,E2 -8794.848} C_VEL
LIN {X 0,Y 446.45,Z 628.875,A -85,B 0,C 180,E1 -8798.245,E2 -8798.245} C_VEL
LIN {X 0,Y 446.459,Z 628.875,A -85,B 0,C 180,E1 -8801.649,E2 -8801.649} C_VEL
LIN {X 0,Y 446.509,Z 628.869,A -85,B 0,C 180,E1 -8804.48,E2 -8804.48} C_VEL
LIN {X 0,Y 446.519,Z 628.867,A -85,B 0,C 180,E1 -8808.193,E2 -8808.193} C_VEL
LIN {X 0,Y 446.602,Z 628.855,A -85,B 0,C 180,E1 -8811.858,E2 -8811.858} C_VEL
LIN {X 0,Y 446.647,Z 628.851,A -85,B 0,C 180,E1 -8814.583,E2 -8814.583} C_VEL
LIN {X 0,Y 446.666,Z 628.849,A -85,B 0,C 180,E1 -8818.197,E2 -8818.197} C_VEL
LIN {X 0,Y 446.795,Z 628.833,A -85,B 0,C 180,E1 -8820,E2 -8820} C_VEL
LIN {X 0,Y 446.711,Z 628.845,A -85,B 0,C 180,E1 -8822.705,E2 -8822.705} C_VEL
LIN {X 0,Y 446.648,Z 628.851,A -85,B 0,C 180,E1 -8826.324,E2 -8826.324} C_VEL
LIN {X 0,Y 446.591,Z 628.859,A -85,B 0,C 180,E1 -8828.142,E2 -8828.142} C_VEL
LIN {X 0,Y 446.493,Z 628.939,A -85,B 0,C 180,E1 -8829.056,E2 -8829.056} C_VEL
LIN {X 0,Y 446.43,Z 632.404,A -85,B 0,C 180,E1 -8831.809,E2 -8831.809} C_VEL
LIN {X 0,Y 446.21,Z 637.26,A -85,B 0,C 180,E1 -8835.531,E2 -8835.531} C_VEL
LIN {X 0,Y 446.023,Z 642.371,A -85,B 0,C 180,E1 -8839.323,E2 -8839.323} C_VEL
LIN {X 0,Y 445.839,Z 646.427,A -85,B 0,C 180,E1 -8842.23,E2 -8842.23} C_VEL
LIN {X 0,Y 445.73,Z 650.616,A -85,B 0,C 180,E1 -8845.196,E2 -8845.196} C_VEL
LIN {X 0,Y 445.582,Z 655.01,A -85,B 0,C 180,E1 -8848.241,E2 -8848.241} C_VEL
LIN {X 0,Y 445.571,Z 655.995,A -85,B 0,C 180,E1 -8848.917,E2 -8848.917} C_VEL
LIN {X 0,Y 448.601,Z 669.749,A -85,B 0,C 180,E1 -8849.472,E2 -8849.472} C_VEL
LIN {X 0,Y 449.549,Z 675.906,A -85,B 0,C 180,E1 -8849.771,E2 -8849.771} C_VEL
LIN {X 0,Y 449.067,Z 687.902,A -85,B 0,C 180,E1 -8850.402,E2 -8850.402} C_VEL
LIN {X 0,Y 448.527,Z 698.632,A -85,B 0,C 180,E1 -8851.137,E2 -8851.137} C_VEL
LIN {X 0,Y 447.943,Z 709.598,A -85,B 0,C 180,E1 -8852.088,E2 -8852.088} C_VEL
LIN {X 0,Y 447.292,Z 720.17,A -85,B 0,C 180,E1 -8853.228,E2 -8853.228} C_VEL
LIN {X 0,Y 446.787,Z 729.53,A -85,B 0,C 180,E1 -8854.492,E2 -8854.492} C_VEL
LIN {X 0,Y 446.302,Z 737.673,A -85,B 0,C 180,E1 -8855.856,E2 -8855.856} C_VEL
LIN {X 0,Y 445.899,Z 744.821,A -85,B 0,C 180,E1 -8857.36,E2 -8857.36} C_VEL
LIN {X 0,Y 445.708,Z 749.207,A -85,B 0,C 180,E1 -8858.524,E2 -8858.524} C_VEL
LIN {X 0,Y 445.568,Z 753.079,A -85,B 0,C 180,E1 -8859.808,E2 -8859.808} C_VEL
LIN {X 0,Y 445.411,Z 756.806,A -85,B 0,C 180,E1 -8861.507,E2 -8861.507} C_VEL
LIN {X 0,Y 445.302,Z 758.55,A -85,B 0,C 180,E1 -8862.739,E2 -8862.739} C_VEL
LIN {X 0,Y 445.267,Z 759.542,A -85,B 0,C 180,E1 -8863.987,E2 -8863.987} C_VEL
LIN {X 0,Y 445.259,Z 759.794,A -85,B 0,C 180,E1 -8865.258,E2 -8865.258} C_VEL
LIN {X 0,Y 445.238,Z 759.252,A -85,B 0,C 180,E1 -8866.561,E2 -8866.561} C_VEL
LIN {X 0,Y 445.329,Z 757.839,A -85,B 0,C 180,E1 -8867.88,E2 -8867.88} C_VEL
LIN {X 0,Y 445.489,Z 754.427,A -85,B 0,C 180,E1 -8869.698,E2 -8869.698} C_VEL
LIN {X 0,Y 445.613,Z 751.259,A -85,B 0,C 180,E1 -8870.886,E2 -8870.886} C_VEL
LIN {X 0,Y 445.818,Z 746.179,A -85,B 0,C 180,E1 -8872.348,E2 -8872.348} C_VEL
LIN {X 0,Y 446.15,Z 739.153,A -85,B 0,C 180,E1 -8873.914,E2 -8873.914} C_VEL
LIN {X 0,Y 446.594,Z 731.772,A -85,B 0,C 180,E1 -8875.217,E2 -8875.217} C_VEL
LIN {X 0,Y 447.122,Z 723.405,A -85,B 0,C 180,E1 -8876.416,E2 -8876.416} C_VEL
LIN {X 0,Y 447.696,Z 713.174,A -85,B 0,C 180,E1 -8877.608,E2 -8877.608} C_VEL
LIN {X 0,Y 448.292,Z 702.806,A -85,B 0,C 180,E1 -8878.582,E2 -8878.582} C_VEL
LIN {X 0,Y 448.828,Z 691.06,A -85,B 0,C 180,E1 -8879.454,E2 -8879.454} C_VEL
LIN {X 0,Y 449.399,Z 679.193,A -85,B 0,C 180,E1 -8880.132,E2 -8880.132} C_VEL
LIN {X 0,Y 449.29,Z 674.008,A -85,B 0,C 180,E1 -8880.382,E2 -8880.382} C_VEL
LIN {X 0,Y 446.908,Z 661.931,A -85,B 0,C 180,E1 -8880.92,E2 -8880.92} C_VEL
LIN {X 0,Y 445.518,Z 655.541,A -85,B 0,C 180,E1 -8881.16,E2 -8881.16} C_VEL
LIN {X 0,Y 445.639,Z 651.31,A -85,B 0,C 180,E1 -8884.018,E2 -8884.018} C_VEL
LIN {X 0,Y 445.728,Z 646.49,A -85,B 0,C 180,E1 -8887.324,E2 -8887.324} C_VEL
LIN {X 0,Y 445.916,Z 641.703,A -85,B 0,C 180,E1 -8890.672,E2 -8890.672} C_VEL
LIN {X 0,Y 445.93,Z 640.964,A -85,B 0,C 180,E1 -8891.191,E2 -8891.191} C_VEL
LIN {X 0,Y 445.297,Z 639.983,A -85,B 0,C 180,E1 -8891.936,E2 -8891.936} C_VEL
LIN {X 0,Y 442.481,Z 638.597,A -85,B 0,C 180,E1 -8893.15,E2 -8893.15} C_VEL
LIN {X 0,Y 440.109,Z 637.519,A -85,B 0,C 180,E1 -8894.131,E2 -8894.131} C_VEL
LIN {X 0,Y 439.125,Z 636.598,A -85,B 0,C 180,E1 -8894.887,E2 -8894.887} C_VEL
LIN {X 0,Y 439.064,Z 636.258,A -85,B 0,C 180,E1 -8895.142,E2 -8895.142} C_VEL
LIN {X 0,Y 439.281,Z 632.407,A -85,B 0,C 180,E1 -8897.995,E2 -8897.995} C_VEL
LIN {X 0,Y 439.278,Z 629.951,A -85,B 0,C 180,E1 -8899.863,E2 -8899.863} C_VEL
LIN {X 0,Y 439.585,Z 629.731,A -85,B 0,C 180,E1 -8902.651,E2 -8902.651} C_VEL
LIN {X 0,Y 439.623,Z 629.725,A -85,B 0,C 180,E1 -8904.495,E2 -8904.495} C_VEL
LIN {X 0,Y 439.639,Z 629.72,A -85,B 0,C 180,E1 -8908.167,E2 -8908.167} C_VEL
LIN {X 0,Y 439.768,Z 629.705,A -85,B 0,C 180,E1 -8910,E2 -8910} C_VEL
LIN {X 0,Y 439.659,Z 629.721,A -85,B 0,C 180,E1 -8912.748,E2 -8912.748} C_VEL
LIN {X 0,Y 439.606,Z 629.726,A -85,B 0,C 180,E1 -8916.425,E2 -8916.425} C_VEL
LIN {X 0,Y 439.353,Z 629.76,A -85,B 0,C 180,E1 -8919.204,E2 -8919.204} C_VEL
LIN {X 0,Y 438.94,Z 630.011,A -85,B 0,C 180,E1 -8921.779,E2 -8921.779} C_VEL
LIN {X 0,Y 438.78,Z 634.919,A -85,B 0,C 180,E1 -8924.849,E2 -8924.849} C_VEL
LIN {X 0,Y 438.674,Z 639.504,A -85,B 0,C 180,E1 -8927.722,E2 -8927.722} C_VEL
LIN {X 0,Y 438.567,Z 644.161,A -85,B 0,C 180,E1 -8930.643,E2 -8930.643} C_VEL
LIN {X 0,Y 438.489,Z 649.476,A -85,B 0,C 180,E1 -8933.994,E2 -8933.994} C_VEL
LIN {X 0,Y 438.407,Z 653.709,A -85,B 0,C 180,E1 -8936.67,E2 -8936.67} C_VEL
LIN {X 0,Y 438.43,Z 655.35,A -85,B 0,C 180,E1 -8937.701,E2 -8937.701} C_VEL
LIN {X 0,Y 441.296,Z 668.889,A -85,B 0,C 180,E1 -8938.23,E2 -8938.23} C_VEL
LIN {X 0,Y 442.601,Z 676.416,A -85,B 0,C 180,E1 -8938.605,E2 -8938.605} C_VEL
LIN {X 0,Y 442.055,Z 688.454,A -85,B 0,C 180,E1 -8939.257,E2 -8939.257} C_VEL
LIN {X 0,Y 441.464,Z 700.279,A -85,B 0,C 180,E1 -8940.097,E2 -8940.097} C_VEL
LIN {X 0,Y 440.834,Z 711.041,A -85,B 0,C 180,E1 -8941.073,E2 -8941.073} C_VEL
LIN {X 0,Y 440.242,Z 721.165,A -85,B 0,C 180,E1 -8942.211,E2 -8942.211} C_VEL
LIN {X 0,Y 439.635,Z 730.216,A -85,B 0,C 180,E1 -8943.47,E2 -8943.47} C_VEL
LIN {X 0,Y 439.19,Z 738.429,A -85,B 0,C 180,E1 -8944.895,E2 -8944.895} C_VEL
LIN {X 0,Y 438.82,Z 745.095,A -85,B 0,C 180,E1 -8946.34,E2 -8946.34} C_VEL
LIN {X 0,Y 438.535,Z 750.587,A -85,B 0,C 180,E1 -8947.877,E2 -8947.877} C_VEL
LIN {X 0,Y 438.358,Z 754.18,A -85,B 0,C 180,E1 -8949.183,E2 -8949.183} C_VEL
LIN {X 0,Y 438.224,Z 756.857,A -85,B 0,C 180,E1 -8950.484,E2 -8950.484} C_VEL
LIN {X 0,Y 438.161,Z 759.184,A -85,B 0,C 180,E1 -8952.35,E2 -8952.35} C_VEL
LIN {X 0,Y 438.157,Z 759.862,A -85,B 0,C 180,E1 -8953.797,E2 -8953.797} C_VEL
LIN {X 0,Y 438.185,Z 759.62,A -85,B 0,C 180,E1 -8955.113,E2 -8955.113} C_VEL
LIN {X 0,Y 438.196,Z 758.608,A -85,B 0,C 180,E1 -8956.397,E2 -8956.397} C_VEL
LIN {X 0,Y 438.274,Z 756.842,A -85,B 0,C 180,E1 -8957.662,E2 -8957.662} C_VEL
LIN {X 0,Y 438.429,Z 754.28,A -85,B 0,C 180,E1 -8958.911,E2 -8958.911} C_VEL
LIN {X 0,Y 438.572,Z 750.531,A -85,B 0,C 180,E1 -8960.28,E2 -8960.28} C_VEL
LIN {X 0,Y 438.845,Z 745.505,A -85,B 0,C 180,E1 -8961.694,E2 -8961.694} C_VEL
LIN {X 0,Y 439.147,Z 738.926,A -85,B 0,C 180,E1 -8963.147,E2 -8963.147} C_VEL
LIN {X 0,Y 439.686,Z 730.601,A -85,B 0,C 180,E1 -8964.605,E2 -8964.605} C_VEL
LIN {X 0,Y 440.254,Z 721.428,A -85,B 0,C 180,E1 -8965.894,E2 -8965.894} C_VEL
LIN {X 0,Y 440.911,Z 711.182,A -85,B 0,C 180,E1 -8967.047,E2 -8967.047} C_VEL
LIN {X 0,Y 441.55,Z 699.872,A -85,B 0,C 180,E1 -8968.07,E2 -8968.07} C_VEL
LIN {X 0,Y 442.147,Z 688.563,A -85,B 0,C 180,E1 -8968.867,E2 -8968.867} C_VEL
LIN {X 0,Y 442.654,Z 677.656,A -85,B 0,C 180,E1 -8969.465,E2 -8969.465} C_VEL
LIN {X 0,Y 441.271,Z 668.368,A -85,B 0,C 180,E1 -8969.925,E2 -8969.925} C_VEL
LIN {X 0,Y 438.462,Z 655.671,A -85,B 0,C 180,E1 -8970.437,E2 -8970.437} C_VEL
LIN {X 0,Y 438.575,Z 650.26,A -85,B 0,C 180,E1 -8973.814,E2 -8973.814} C_VEL
LIN {X 0,Y 438.6,Z 644.494,A -85,B 0,C 180,E1 -8977.383,E2 -8977.383} C_VEL
LIN {X 0,Y 438.738,Z 638.723,A -85,B 0,C 180,E1 -8980.924,E2 -8980.924} C_VEL
LIN {X 0,Y 438.825,Z 633.152,A -85,B 0,C 180,E1 -8984.201,E2 -8984.201} C_VEL
LIN {X 0,Y 438.916,Z 629.818,A -85,B 0,C 180,E1 -8986.221,E2 -8986.221} C_VEL
LIN {X 0,Y 439.313,Z 629.766,A -85,B 0,C 180,E1 -8988.932,E2 -8988.932} C_VEL
LIN {X 0,Y 439.542,Z 629.737,A -85,B 0,C 180,E1 -8991.726,E2 -8991.726} C_VEL
LIN {X 0,Y 439.619,Z 629.727,A -85,B 0,C 180,E1 -8994.496,E2 -8994.496} C_VEL
LIN {X 0,Y 439.632,Z 629.726,A -85,B 0,C 180,E1 -8998.168,E2 -8998.168} C_VEL
LIN {X 0,Y 439.761,Z 629.709,A -85,B 0,C 180,E1 -9000,E2 -9000} C_VEL
LIN {X 0,Y 439.653,Z 629.722,A -85,B 0,C 180,E1 -9002.749,E2 -9002.749} C_VEL
LIN {X 0,Y 439.615,Z 629.728,A -85,B 0,C 180,E1 -9006.425,E2 -9006.425} C_VEL
LIN {X 0,Y 439.497,Z 629.741,A -85,B 0,C 180,E1 -9009.202,E2 -9009.202} C_VEL
LIN {X 0,Y 439.461,Z 629.746,A -85,B 0,C 180,E1 -9012.938,E2 -9012.938} C_VEL
LIN {X 0,Y 439.443,Z 629.747,A -85,B 0,C 180,E1 -9016.349,E2 -9016.349} C_VEL
LIN {X 0,Y 439.399,Z 629.753,A -85,B 0,C 180,E1 -9019.626,E2 -9019.626} C_VEL
LIN {X 0,Y 439.362,Z 629.758,A -85,B 0,C 180,E1 -9022.576,E2 -9022.576} C_VEL
LIN {X 0,Y 439.402,Z 629.753,A -85,B 0,C 180,E1 -9025.585,E2 -9025.585} C_VEL
LIN {X 0,Y 439.422,Z 629.748,A -85,B 0,C 180,E1 -9028.673,E2 -9028.673} C_VEL
LIN {X 0,Y 439.372,Z 629.757,A -85,B 0,C 180,E1 -9031.861,E2 -9031.861} C_VEL
LIN {X 0,Y 439.398,Z 629.754,A -85,B 0,C 180,E1 -9035.156,E2 -9035.156} C_VEL
LIN {X 0,Y 439.386,Z 629.756,A -85,B 0,C 180,E1 -9038.595,E2 -9038.595} C_VEL
LIN {X 0,Y 439.386,Z 629.756,A -85,B 0,C 180,E1 -9041.257,E2 -9041.257} C_VEL
LIN {X 0,Y 439.399,Z 629.754,A -85,B 0,C 180,E1 -9044.73,E2 -9044.73} C_VEL
LIN {X 0,Y 439.394,Z 629.755,A -85,B 0,C 180,E1 -9047.796,E2 -9047.796} C_VEL
LIN {X 0,Y 439.467,Z 629.907,A -85,B 0,C 180,E1 -9050.077,E2 -9050.077} C_VEL
LIN {X 0,Y 440.279,Z 635.153,A -85,B 0,C 180,E1 -9052.952,E2 -9052.952} C_VEL
LIN {X 0,Y 440.524,Z 638.984,A -85,B 0,C 180,E1 -9054.948,E2 -9054.948} C_VEL
LIN {X 0,Y 440.114,Z 645.552,A -85,B 0,C 180,E1 -9058.2,E2 -9058.2} C_VEL
LIN {X 0,Y 439.774,Z 652.485,A -85,B 0,C 180,E1 -9061.517,E2 -9061.517} C_VEL
LIN {X 0,Y 439.396,Z 659.851,A -85,B 0,C 180,E1 -9064.922,E2 -9064.922} C_VEL
LIN {X 0,Y 439.1,Z 667.566,A -85,B 0,C 180,E1 -9068.4,E2 -9068.4} C_VEL
LIN {X 0,Y 438.829,Z 674.172,A -85,B 0,C 180,E1 -9071.319,E2 -9071.319} C_VEL
LIN {X 0,Y 438.757,Z 679.467,A -85,B 0,C 180,E1 -9073.617,E2 -9073.617} C_VEL
LIN {X 0,Y 440.976,Z 692.858,A -85,B 0,C 180,E1 -9074.085,E2 -9074.085} C_VEL
LIN {X 0,Y 442.415,Z 703.039,A -85,B 0,C 180,E1 -9074.569,E2 -9074.569} C_VEL
LIN {X 0,Y 441.821,Z 715.373,A -85,B 0,C 180,E1 -9075.256,E2 -9075.256} C_VEL
LIN {X 0,Y 441.231,Z 726.485,A -85,B 0,C 180,E1 -9076.06,E2 -9076.06} C_VEL
LIN {X 0,Y 440.628,Z 737.86,A -85,B 0,C 180,E1 -9077.098,E2 -9077.098} C_VEL
LIN {X 0,Y 439.975,Z 747.91,A -85,B 0,C 180,E1 -9078.249,E2 -9078.249} C_VEL
LIN {X 0,Y 439.392,Z 757.644,A -85,B 0,C 180,E1 -9079.634,E2 -9079.634} C_VEL
LIN {X 0,Y 438.983,Z 765.418,A -85,B 0,C 180,E1 -9081.02,E2 -9081.02} C_VEL
LIN {X 0,Y 438.592,Z 772.559,A -85,B 0,C 180,E1 -9082.635,E2 -9082.635} C_VEL
LIN {X 0,Y 438.416,Z 777.062,A -85,B 0,C 180,E1 -9083.938,E2 -9083.938} C_VEL
LIN {X 0,Y 438.354,Z 780.952,A -85,B 0,C 180,E1 -9085.402,E2 -9085.402} C_VEL
LIN {X 0,Y 438.286,Z 782.826,A -85,B 0,C 180,E1 -9086.323,E2 -9086.323} C_VEL
LIN {X 0,Y 438.331,Z 784.234,A -85,B 0,C 180,E1 -9087.243,E2 -9087.243} C_VEL
LIN {X 0,Y 438.251,Z 785.839,A -85,B 0,C 180,E1 -9089.082,E2 -9089.082} C_VEL
LIN {X 0,Y 438.253,Z 786.053,A -85,B 0,C 180,E1 -9090,E2 -9090} C_VEL
LIN {X 0,Y 438.251,Z 785.831,A -85,B 0,C 180,E1 -9090.919,E2 -9090.919} C_VEL
LIN {X 0,Y 438.331,Z 784.204,A -85,B 0,C 180,E1 -9092.757,E2 -9092.757} C_VEL
LIN {X 0,Y 438.287,Z 782.788,A -85,B 0,C 180,E1 -9093.678,E2 -9093.678} C_VEL
LIN {X 0,Y 438.404,Z 779.821,A -85,B 0,C 180,E1 -9095.059,E2 -9095.059} C_VEL
LIN {X 0,Y 438.506,Z 775.805,A -85,B 0,C 180,E1 -9096.442,E2 -9096.442} C_VEL
LIN {X 0,Y 438.727,Z 769.63,A -85,B 0,C 180,E1 -9098.058,E2 -9098.058} C_VEL
LIN {X 0,Y 439.075,Z 762.892,A -85,B 0,C 180,E1 -9099.443,E2 -9099.443} C_VEL
LIN {X 0,Y 439.532,Z 754.549,A -85,B 0,C 180,E1 -9100.829,E2 -9100.829} C_VEL
LIN {X 0,Y 440.118,Z 745.995,A -85,B 0,C 180,E1 -9101.981,E2 -9101.981} C_VEL
LIN {X 0,Y 440.671,Z 735.921,A -85,B 0,C 180,E1 -9103.089,E2 -9103.089} C_VEL
LIN {X 0,Y 441.261,Z 725.034,A -85,B 0,C 180,E1 -9104.057,E2 -9104.057} C_VEL
LIN {X 0,Y 441.916,Z 713.649,A -85,B 0,C 180,E1 -9104.859,E2 -9104.859} C_VEL
LIN {X 0,Y 442.297,Z 701.977,A -85,B 0,C 180,E1 -9105.495,E2 -9105.495} C_VEL
LIN {X 0,Y 440.278,Z 687.957,A -85,B 0,C 180,E1 -9106.128,E2 -9106.128} C_VEL
LIN {X 0,Y 438.717,Z 678.991,A -85,B 0,C 180,E1 -9106.437,E2 -9106.437} C_VEL
LIN {X 0,Y 438.971,Z 670.482,A -85,B 0,C 180,E1 -9110.134,E2 -9110.134} C_VEL
LIN {X 0,Y 439.149,Z 663.87,A -85,B 0,C 180,E1 -9113.085,E2 -9113.085} C_VEL
LIN {X 0,Y 439.396,Z 658.39,A -85,B 0,C 180,E1 -9115.586,E2 -9115.586} C_VEL
LIN {X 0,Y 439.721,Z 651.881,A -85,B 0,C 180,E1 -9118.652,E2 -9118.652} C_VEL
LIN {X 0,Y 440.093,Z 645.462,A -85,B 0,C 180,E1 -9121.802,E2 -9121.802} C_VEL
LIN {X 0,Y 440.481,Z 640.196,A -85,B 0,C 180,E1 -9124.501,E2 -9124.501} C_VEL
LIN {X 0,Y 440.515,Z 637.083,A -85,B 0,C 180,E1 -9126.178,E2 -9126.178} C_VEL
LIN {X 0,Y 439.966,Z 633.015,A -85,B 0,C 180,E1 -9128.535,E2 -9128.535} C_VEL
LIN {X 0,Y 439.408,Z 629.755,A -85,B 0,C 180,E1 -9130.61,E2 -9130.61} C_VEL
